REGION Network 34: CONVEYORS
   // FC71 = 0 IN + 0 OUT; FC72 = 0 IN + 1 OUT; FC73 = 0 IN + 2 OUT; FC74 = 0 IN + 3 OUT; FC75 = 0 IN + 4 OUT
   // FC76 = 1 IN + 0 OUT; FC77 = 1 IN + 1 OUT; FC78 = 1 IN + 2 OUT; FC79 = 1 IN + 3 OUT
   // FC80 = 2 IN + 0 OUT; FC81 = 2 IN + 1 OUT; FC82 = 2 IN + 2 OUT
   // FC83 = 3 IN + 0 OUT; FC84 = 3 IN + 1 OUT
   // FC85 = 4 IN + 0 OUT
   // FC86 = SPECIAL
   RUNG wire#powerrail
      Contact( "On" )
      wire#w1
      "FC31_ConveyorInverter"()
   END_RUNG
   RUNG wire#w1
      I_Contact( "On" )
      "FC32_ConveyorInverter_REV"()
   END_RUNG
   RUNG wire#w1
      { S7_Templates := "SrcType := Int" } EQ_Contact(in1 := "DB50_Config".Sel10_Conv, in2 := 16)
      "FC86_Conveyor_5_IN_3_OUT"()
   END_RUNG
   RUNG wire#w1
      { S7_Templates := "SrcType := Int" } EQ_Contact(in1 := "DB50_Config".Sel10_Conv, in2 := 1)
      "FC71_Conveyor_0_IN_0_OUT"()
   END_RUNG
   RUNG wire#w1
      { S7_Templates := "SrcType := Int" } EQ_Contact(in1 := "DB50_Config".Sel10_Conv, in2 := 2)
      "FC72_Conveyor_0_IN_1_OUT"()
   END_RUNG
   RUNG wire#w1
      { S7_Templates := "SrcType := Int" } EQ_Contact(in1 := "DB50_Config".Sel10_Conv, in2 := 7)
      wire#w2
      "FC77_Conveyor_1_IN_1_OUT"()
   END_RUNG
   RUNG wire#w2
      I_Contact( "On" )
      "FC78_Conveyor_1_IN_1_OUT_REVERSE"()
   END_RUNG
   RUNG wire#w1
      { S7_Templates := "SrcType := Int" } EQ_Contact(in1 := "DB50_Config".Sel10_Conv, in2 := 12)
      "FC82_Conveyor_2_IN_2_OUT"()
   END_RUNG
   // the same network as SCL:
   #_w1 := "On";
   IF #_w1 THEN "FC31_ConveyorInverter"(); END_IF;
   IF #_w1 AND NOT "On" THEN "FC32_ConveyorInverter_REV"(); END_IF;
   IF #_w1 AND ("DB50_Config".Sel10_Conv = 16) THEN "FC86_Conveyor_5_IN_3_OUT"(); END_IF;
   IF #_w1 AND ("DB50_Config".Sel10_Conv = 1) THEN "FC71_Conveyor_0_IN_0_OUT"(); END_IF;
   IF #_w1 AND ("DB50_Config".Sel10_Conv = 2) THEN "FC72_Conveyor_0_IN_1_OUT"(); END_IF;
   #_w2 := #_w1 AND ("DB50_Config".Sel10_Conv = 7);
   IF #_w2 THEN "FC77_Conveyor_1_IN_1_OUT"(); END_IF;
   IF #_w2 AND NOT "On" THEN "FC78_Conveyor_1_IN_1_OUT_REVERSE"(); END_IF;
   IF #_w1 AND ("DB50_Config".Sel10_Conv = 12) THEN "FC82_Conveyor_2_IN_2_OUT"(); END_IF;
END_REGION

REGION Network 35: BARRIERS
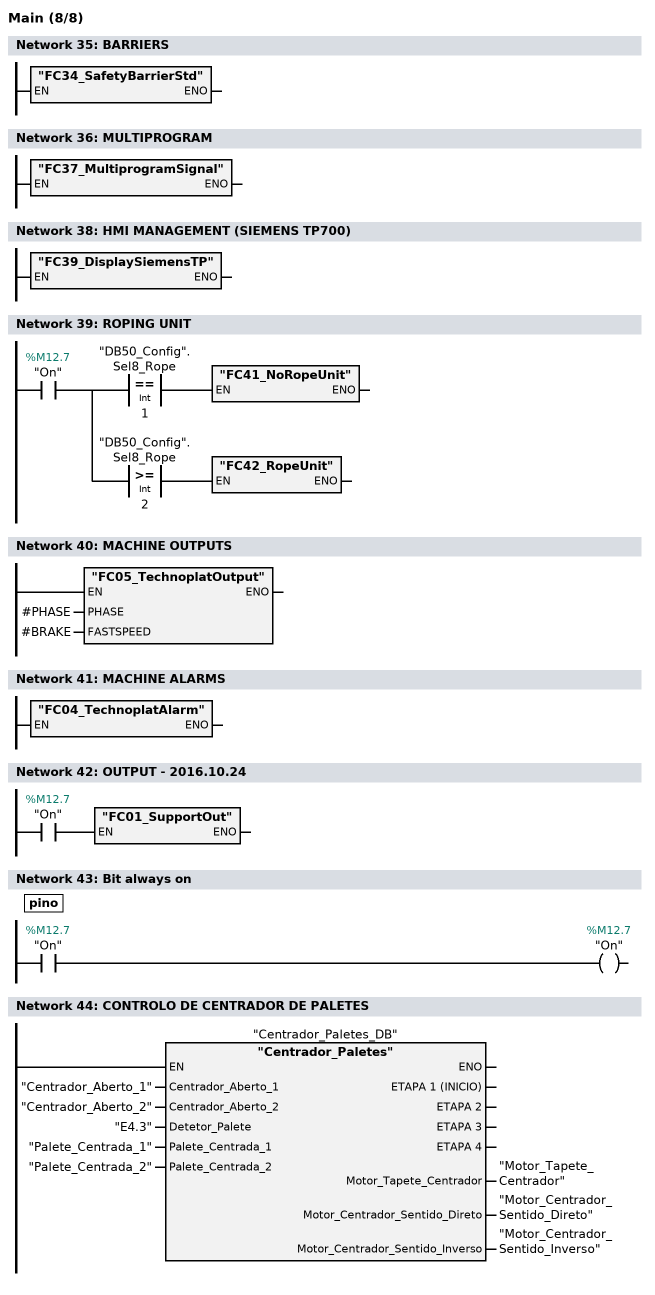
   RUNG wire#powerrail
      "FC34_SafetyBarrierStd"()
   END_RUNG
   // the same network as SCL:
   "FC34_SafetyBarrierStd"();
END_REGION

REGION Network 36: MULTIPROGRAM
   RUNG wire#powerrail
      "FC37_MultiprogramSignal"()
   END_RUNG
   // the same network as SCL:
   "FC37_MultiprogramSignal"();
END_REGION

REGION Network 37: Incomplete pallet
END_REGION

REGION Network 38: HMI MANAGEMENT (SIEMENS TP700)
   RUNG wire#powerrail
      "FC39_DisplaySiemensTP"()
   END_RUNG
   // the same network as SCL:
   "FC39_DisplaySiemensTP"();
END_REGION

REGION Network 39: ROPING UNIT
   RUNG wire#powerrail
      Contact( "On" )
      wire#w1
      { S7_Templates := "SrcType := Int" } EQ_Contact(in1 := "DB50_Config".Sel8_Rope, in2 := 1)
      "FC41_NoRopeUnit"()
   END_RUNG
   RUNG wire#w1
      { S7_Templates := "SrcType := Int" } GE_Contact(in1 := "DB50_Config".Sel8_Rope, in2 := 2)
      "FC42_RopeUnit"()
   END_RUNG
   // the same network as SCL:
   #_w1 := "On";
   IF "On" AND ("DB50_Config".Sel8_Rope = 1) THEN "FC41_NoRopeUnit"(); END_IF;
   IF #_w1 AND ("DB50_Config".Sel8_Rope >= 2) THEN "FC42_RopeUnit"(); END_IF;
END_REGION

REGION Network 40: MACHINE OUTPUTS
   RUNG wire#powerrail
      "FC05_TechnoplatOutput"(PHASE := #PHASE, FASTSPEED := #BRAKE)
   END_RUNG
   // the same network as SCL:
   "FC05_TechnoplatOutput"(PHASE := #PHASE, FASTSPEED := #BRAKE);
END_REGION

REGION Network 41: MACHINE ALARMS
   RUNG wire#powerrail
      "FC04_TechnoplatAlarm"()
   END_RUNG
   // the same network as SCL:
   "FC04_TechnoplatAlarm"();
END_REGION

REGION Network 42: OUTPUT - 2016.10.24
   RUNG wire#powerrail
      Contact( "On" )
      "FC01_SupportOut"()
   END_RUNG
   // the same network as SCL:
   IF "On" THEN "FC01_SupportOut"(); END_IF;
END_REGION

REGION Network 43: Bit always on
   Label( pino )
   RUNG wire#powerrail
      Contact( "On" )
      Coil( "On" )
   END_RUNG
   // the same network as SCL:
   pino:
   "On" := "On";
END_REGION

REGION Network 44: CONTROLO DE CENTRADOR DE PALETES
   RUNG wire#powerrail
      "Centrador_Paletes_DB"(Centrador_Aberto_1 := "Centrador_Aberto_1", Centrador_Aberto_2 := "Centrador_Aberto_2", Detetor_Palete := "E4.3", Palete_Centrada_1 := "Palete_Centrada_1", Palete_Centrada_2 := "Palete_Centrada_2", "ETAPA 1 (INICIO)" =>, "ETAPA 2" =>, "ETAPA 3" =>, "ETAPA 4" =>, Motor_Tapete_Centrador => "Motor_Tapete_Centrador", Motor_Centrador_Sentido_Direto => "Motor_Centrador_Sentido_Direto", Motor_Centrador_Sentido_Inverso => "Motor_Centrador_Sentido_Inverso")
   END_RUNG
   // the same network as SCL:
   "Centrador_Paletes_DB"(Centrador_Aberto_1 := "Centrador_Aberto_1",   // "Centrador_Paletes"
                          Centrador_Aberto_2 := "Centrador_Aberto_2",
                          Detetor_Palete := "E4.3",
                          Palete_Centrada_1 := "Palete_Centrada_1",
                          Palete_Centrada_2 := "Palete_Centrada_2",
                          Motor_Tapete_Centrador => "Motor_Tapete_Centrador",
                          Motor_Centrador_Sentido_Direto => "Motor_Centrador_Sentido_Direto",
                          Motor_Centrador_Sentido_Inverso => "Motor_Centrador_Sentido_Inverso");
END_REGION
END_ORGANIZATION_BLOCK

FUNCTION_BLOCK "Modbus"   // FB20, FBD
{ S7_Optimized_Access := 'FALSE' }
VERSION : 0.1
// stored: AutoNumber false, IsIECCheckEnabled false, SetENOAutomatically false, UDAEnableTagReadback false
   VAR_INPUT
      BAUDRATE : UDInt := 115200;
      HW_ID : PORT := 272;
      RESP_TO : UInt := 1000;
      CYCLIC_PROCESSING : Bool := true;
      MB_ADDR : UInt := 8;
      DATA_AD_R : UDInt := 40001;
      DATA_AD_W : UDInt := 40006;
      DATA_LEN_R : UInt := 5;
      DATA_LEN_W : UInt := 5;
      ReadOnly : Bool := 1;   // Read only (1)
   END_VAR
   VAR_OUTPUT
      ERROR : Bool;
      ERROR_INFO : Struct
         drive_number : USInt;
         "step" : USInt;
         STATUS : Word;
      END_STRUCT;
   END_VAR
   VAR_IN_OUT
      ReadDone_0 : Bool;   // Read done for prestretch board (1)
      DT_PTR_IN : Variant;
      DT_PTR_OUT : Variant;
   END_VAR
   VAR DB_SPECIFIC
      drive_index : USInt := 1;
      "step" : USInt := 0;
      REQ : Bool;
      extended_restart : Bool;
      start_internal : Bool;
   END_VAR
   VAR
      MB_COMM_LOAD_Instance { S7_SetPoint := 'True'} : MB_COMM_LOAD;
      MB_MASTER_Instance { S7_SetPoint := 'True'} : MB_MASTER;
   END_VAR
   VAR_TEMP
      _DONE : Bool;
      _ERROR : Bool;
      _STATUS : Word;
      _cyclic_processing : Bool;
   END_VAR
   VAR_TEMP   // added for the SCL form of the ladder/FBD networks
      _w1 : Bool;
      _w2 : Bool;
      _w3 : Bool;
   END_VAR
BEGIN

REGION Network 1: First cycle
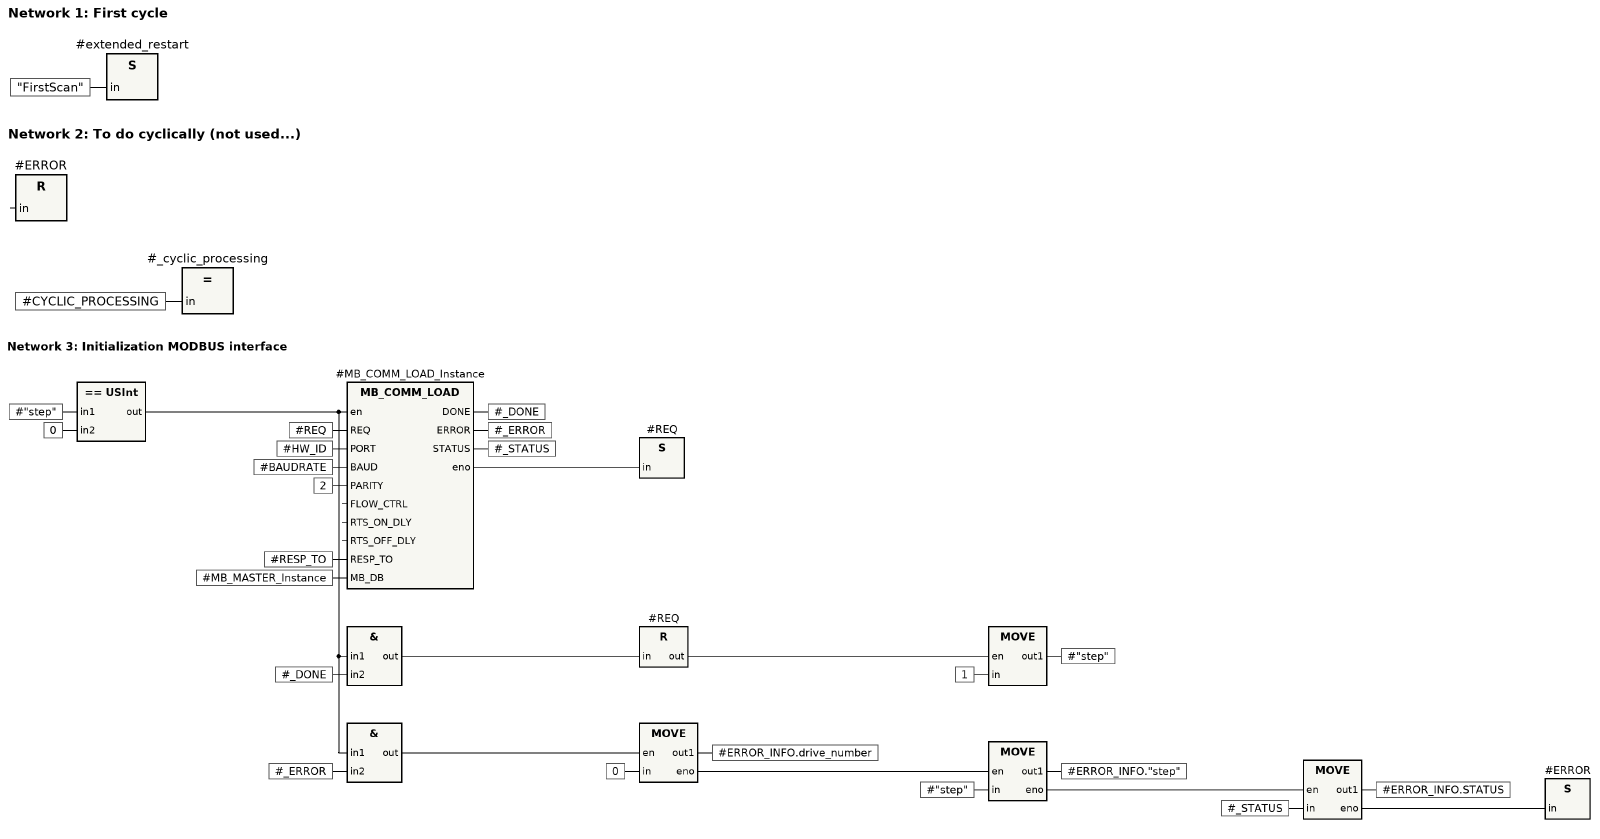
   IF "FirstScan" THEN #extended_restart := TRUE; END_IF;
END_REGION

REGION Network 2: To do cyclically (not used...)
   #ERROR := FALSE;
   #_cyclic_processing := #CYCLIC_PROCESSING;
END_REGION

REGION Network 3: Initialization MODBUS interface
   // ENO of a box is taken as its EN; it also drops when the box reports an error
   #_w1 := #"step" = 0;
   #MB_COMM_LOAD_Instance(EN := #_w1,   // MB_COMM_LOAD
                          REQ := #REQ,
                          PORT := #HW_ID,
                          BAUD := #BAUDRATE,
                          PARITY := 2,
                          RESP_TO := #RESP_TO,
                          MB_DB := #MB_MASTER_Instance,
                          DONE => #_DONE,
                          ERROR => #_ERROR,
                          STATUS => #_STATUS,
                          ENO => #_w2);
   IF #_w2 THEN #REQ := TRUE; END_IF;
   IF #_w1 AND #_DONE THEN
       #REQ := FALSE;
       #"step" := 1;
   END_IF;
   IF #_w1 AND #_ERROR THEN
       #ERROR_INFO.drive_number := 0;
       #ERROR_INFO."step" := #"step";
       #ERROR_INFO.STATUS := #_STATUS;
       #ERROR := TRUE;
   END_IF;
END_REGION

REGION Network 4: READ
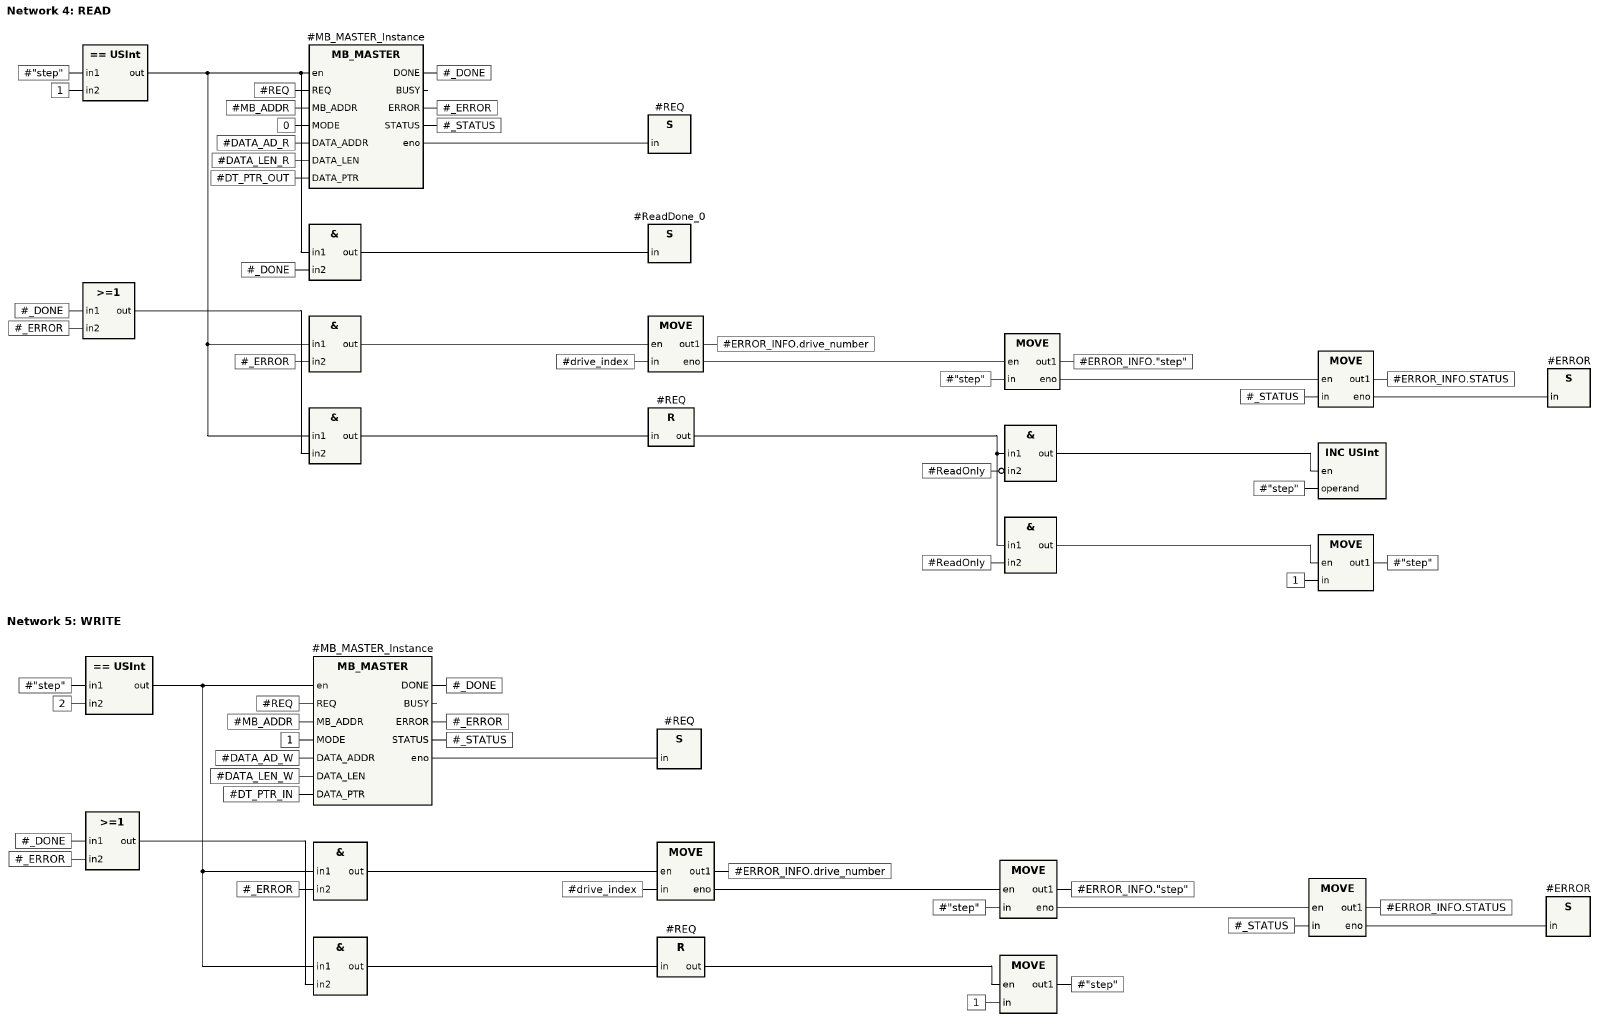
   // ENO of a box is taken as its EN; it also drops when the box reports an error
   #_w1 := #"step" = 1;
   #MB_MASTER_Instance(EN := #_w1,   // MB_MASTER
                       REQ := #REQ,
                       MB_ADDR := #MB_ADDR,
                       MODE := 0,
                       DATA_ADDR := #DATA_AD_R,
                       DATA_LEN := #DATA_LEN_R,
                       DATA_PTR := #DT_PTR_OUT,
                       DONE => #_DONE,
                       ERROR => #_ERROR,
                       STATUS => #_STATUS,
                       ENO => #_w2);
   IF #_w2 THEN #REQ := TRUE; END_IF;
   IF #_w1 AND #_DONE THEN #ReadDone_0 := TRUE; END_IF;
   IF #_w1 AND #_ERROR THEN
       #ERROR_INFO.drive_number := #drive_index;
       #ERROR_INFO."step" := #"step";
       #ERROR_INFO.STATUS := #_STATUS;
       #ERROR := TRUE;
   END_IF;
   #_w3 := #_w1 AND (#_DONE OR #_ERROR);
   IF #_w3 THEN #REQ := FALSE; END_IF;
   IF #_w3 AND NOT #ReadOnly THEN #"step" := #"step" + 1; END_IF;
   IF #_w3 AND #ReadOnly THEN #"step" := 1; END_IF;
END_REGION

REGION Network 5: WRITE
   // ENO of a box is taken as its EN; it also drops when the box reports an error
   #_w1 := #"step" = 2;
   #MB_MASTER_Instance(EN := #_w1,   // MB_MASTER
                       REQ := #REQ,
                       MB_ADDR := #MB_ADDR,
                       MODE := 1,
                       DATA_ADDR := #DATA_AD_W,
                       DATA_LEN := #DATA_LEN_W,
                       DATA_PTR := #DT_PTR_IN,
                       DONE => #_DONE,
                       ERROR => #_ERROR,
                       STATUS => #_STATUS,
                       ENO => #_w2);
   IF #_w2 THEN #REQ := TRUE; END_IF;
   IF #_w1 AND #_ERROR THEN
       #ERROR_INFO.drive_number := #drive_index;
       #ERROR_INFO."step" := #"step";
       #ERROR_INFO.STATUS := #_STATUS;
       #ERROR := TRUE;
   END_IF;
   IF #_w1 AND (#_DONE OR #_ERROR) THEN
       #REQ := FALSE;
       #"step" := 1;
   END_IF;
END_REGION
END_FUNCTION_BLOCK

FUNCTION "FC81_Optional" : Void   // FC81, LAD
TITLE = Optional
{ S7_Optimized_Access := 'TRUE' }
VERSION : 0.1
// stored: AutoNumber false, IsIECCheckEnabled false, SetENOAutomatically false, UDAEnableTagReadback false
BEGIN

REGION Network 1: Signal Automatic
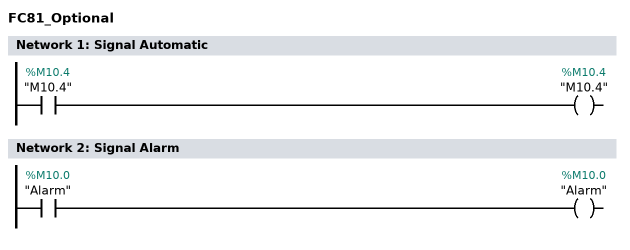
   RUNG wire#powerrail
      Contact( "M10.4" )
      Coil( "M10.4" )
   END_RUNG
   // the same network as SCL:
   "M10.4" := "M10.4";
END_REGION

REGION Network 2: Signal Alarm
   RUNG wire#powerrail
      Contact( "Alarm" )
      Coil( "Alarm" )
   END_RUNG
   // the same network as SCL:
   "Alarm" := "Alarm";
END_REGION
END_FUNCTION

FUNCTION "FC90_PageManagement" : Void   // FC90, LAD
{ S7_Optimized_Access := 'FALSE' }
VERSION : 0.1
// stored: AutoNumber false, IsIECCheckEnabled false, SetENOAutomatically false, UDAEnableTagReadback false
   VAR_TEMP
      CurrentPage : Int;
      PageBkwRequest : Int;
      PageFwRequest : Int;
   END_VAR
   VAR_TEMP   // added for the SCL form of the ladder/FBD networks
      _w1 : Bool;
   END_VAR
BEGIN

REGION Network 1
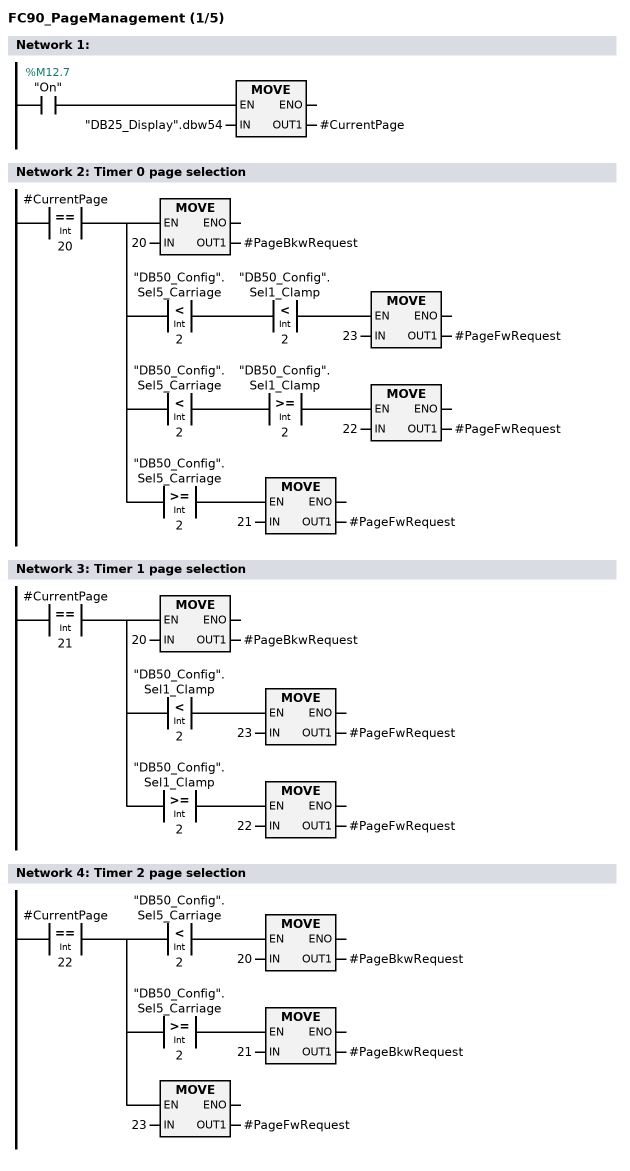
   RUNG wire#powerrail
      Contact( "On" )
      { S7_GenerateENO := "TRUE" } Move(in := "DB25_Display".dbw54, out1 => #CurrentPage)
   END_RUNG
   // the same network as SCL:
   IF "On" THEN #CurrentPage := "DB25_Display".dbw54; END_IF;
END_REGION

REGION Network 2: Timer 0 page selection
   RUNG wire#powerrail
      { S7_Templates := "SrcType := Int" } EQ_Contact(in1 := #CurrentPage, in2 := 20)
      wire#w1
      { S7_GenerateENO := "TRUE" } Move(in := 20, out1 => #PageBkwRequest)
   END_RUNG
   RUNG wire#w1
      { S7_Templates := "SrcType := Int" } LT_Contact(in1 := "DB50_Config".Sel5_Carriage, in2 := 2)
      { S7_Templates := "SrcType := Int" } LT_Contact(in1 := "DB50_Config".Sel1_Clamp, in2 := 2)
      { S7_GenerateENO := "TRUE" } Move(in := 23, out1 => #PageFwRequest)
   END_RUNG
   RUNG wire#w1
      { S7_Templates := "SrcType := Int" } LT_Contact(in1 := "DB50_Config".Sel5_Carriage, in2 := 2)
      { S7_Templates := "SrcType := Int" } GE_Contact(in1 := "DB50_Config".Sel1_Clamp, in2 := 2)
      { S7_GenerateENO := "TRUE" } Move(in := 22, out1 => #PageFwRequest)
   END_RUNG
   RUNG wire#w1
      { S7_Templates := "SrcType := Int" } GE_Contact(in1 := "DB50_Config".Sel5_Carriage, in2 := 2)
      { S7_GenerateENO := "TRUE" } Move(in := 21, out1 => #PageFwRequest)
   END_RUNG
   // the same network as SCL:
   #_w1 := #CurrentPage = 20;
   IF #_w1 THEN #PageBkwRequest := 20; END_IF;
   IF #_w1 AND ("DB50_Config".Sel5_Carriage < 2) AND ("DB50_Config".Sel1_Clamp < 2) THEN
       #PageFwRequest := 23;
   END_IF;
   IF #_w1 AND ("DB50_Config".Sel5_Carriage < 2) AND ("DB50_Config".Sel1_Clamp >= 2) THEN
       #PageFwRequest := 22;
   END_IF;
   IF #_w1 AND ("DB50_Config".Sel5_Carriage >= 2) THEN #PageFwRequest := 21; END_IF;
END_REGION

REGION Network 3: Timer 1 page selection
   RUNG wire#powerrail
      { S7_Templates := "SrcType := Int" } EQ_Contact(in1 := #CurrentPage, in2 := 21)
      wire#w1
      { S7_GenerateENO := "TRUE" } Move(in := 20, out1 => #PageBkwRequest)
   END_RUNG
   RUNG wire#w1
      { S7_Templates := "SrcType := Int" } LT_Contact(in1 := "DB50_Config".Sel1_Clamp, in2 := 2)
      { S7_GenerateENO := "TRUE" } Move(in := 23, out1 => #PageFwRequest)
   END_RUNG
   RUNG wire#w1
      { S7_Templates := "SrcType := Int" } GE_Contact(in1 := "DB50_Config".Sel1_Clamp, in2 := 2)
      { S7_GenerateENO := "TRUE" } Move(in := 22, out1 => #PageFwRequest)
   END_RUNG
   // the same network as SCL:
   #_w1 := #CurrentPage = 21;
   IF #_w1 THEN #PageBkwRequest := 20; END_IF;
   IF #_w1 AND ("DB50_Config".Sel1_Clamp < 2) THEN #PageFwRequest := 23; END_IF;
   IF #_w1 AND ("DB50_Config".Sel1_Clamp >= 2) THEN #PageFwRequest := 22; END_IF;
END_REGION

REGION Network 4: Timer 2 page selection
   RUNG wire#powerrail
      { S7_Templates := "SrcType := Int" } EQ_Contact(in1 := #CurrentPage, in2 := 22)
      wire#w1
      { S7_Templates := "SrcType := Int" } LT_Contact(in1 := "DB50_Config".Sel5_Carriage, in2 := 2)
      { S7_GenerateENO := "TRUE" } Move(in := 20, out1 => #PageBkwRequest)
   END_RUNG
   RUNG wire#w1
      { S7_Templates := "SrcType := Int" } GE_Contact(in1 := "DB50_Config".Sel5_Carriage, in2 := 2)
      { S7_GenerateENO := "TRUE" } Move(in := 21, out1 => #PageBkwRequest)
   END_RUNG
   RUNG wire#w1
      { S7_GenerateENO := "TRUE" } Move(in := 23, out1 => #PageFwRequest)
   END_RUNG
   // the same network as SCL:
   #_w1 := #CurrentPage = 22;
   IF #_w1 AND ("DB50_Config".Sel5_Carriage < 2) THEN #PageBkwRequest := 20; END_IF;
   IF #_w1 AND ("DB50_Config".Sel5_Carriage >= 2) THEN #PageBkwRequest := 21; END_IF;
   IF #_w1 THEN #PageFwRequest := 23; END_IF;
END_REGION

REGION Network 5: Timer 3 page selection
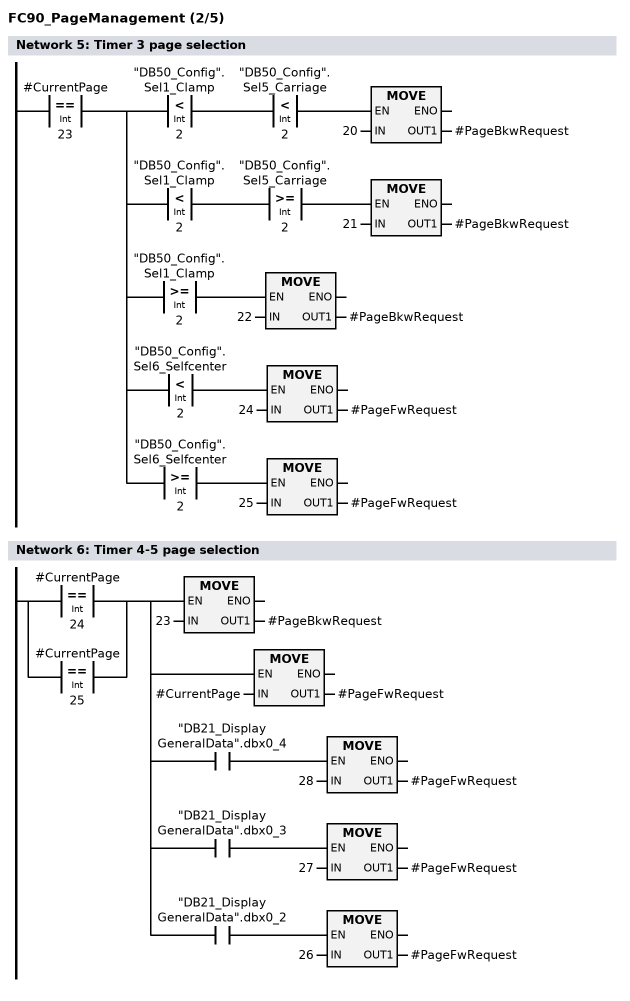
   RUNG wire#powerrail
      { S7_Templates := "SrcType := Int" } EQ_Contact(in1 := #CurrentPage, in2 := 23)
      wire#w1
      { S7_Templates := "SrcType := Int" } LT_Contact(in1 := "DB50_Config".Sel1_Clamp, in2 := 2)
      { S7_Templates := "SrcType := Int" } LT_Contact(in1 := "DB50_Config".Sel5_Carriage, in2 := 2)
      { S7_GenerateENO := "TRUE" } Move(in := 20, out1 => #PageBkwRequest)
   END_RUNG
   RUNG wire#w1
      { S7_Templates := "SrcType := Int" } LT_Contact(in1 := "DB50_Config".Sel1_Clamp, in2 := 2)
      { S7_Templates := "SrcType := Int" } GE_Contact(in1 := "DB50_Config".Sel5_Carriage, in2 := 2)
      { S7_GenerateENO := "TRUE" } Move(in := 21, out1 => #PageBkwRequest)
   END_RUNG
   RUNG wire#w1
      { S7_Templates := "SrcType := Int" } GE_Contact(in1 := "DB50_Config".Sel1_Clamp, in2 := 2)
      { S7_GenerateENO := "TRUE" } Move(in := 22, out1 => #PageBkwRequest)
   END_RUNG
   RUNG wire#w1
      { S7_Templates := "SrcType := Int" } LT_Contact(in1 := "DB50_Config".Sel6_Selfcenter, in2 := 2)
      { S7_GenerateENO := "TRUE" } Move(in := 24, out1 => #PageFwRequest)
   END_RUNG
   RUNG wire#w1
      { S7_Templates := "SrcType := Int" } GE_Contact(in1 := "DB50_Config".Sel6_Selfcenter, in2 := 2)
      { S7_GenerateENO := "TRUE" } Move(in := 25, out1 => #PageFwRequest)
   END_RUNG
   // the same network as SCL:
   #_w1 := #CurrentPage = 23;
   IF #_w1 AND ("DB50_Config".Sel1_Clamp < 2) AND ("DB50_Config".Sel5_Carriage < 2) THEN
       #PageBkwRequest := 20;
   END_IF;
   IF #_w1 AND ("DB50_Config".Sel1_Clamp < 2) AND ("DB50_Config".Sel5_Carriage >= 2) THEN
       #PageBkwRequest := 21;
   END_IF;
   IF #_w1 AND ("DB50_Config".Sel1_Clamp >= 2) THEN #PageBkwRequest := 22; END_IF;
   IF #_w1 AND ("DB50_Config".Sel6_Selfcenter < 2) THEN #PageFwRequest := 24; END_IF;
   IF #_w1 AND ("DB50_Config".Sel6_Selfcenter >= 2) THEN #PageFwRequest := 25; END_IF;
END_REGION

REGION Network 6: Timer 4-5 page selection
   RUNG wire#powerrail
      { S7_Templates := "SrcType := Int" } EQ_Contact(in1 := #CurrentPage, in2 := 24)
      wire#w1
      { S7_GenerateENO := "TRUE" } Move(in := 23, out1 => #PageBkwRequest)
   END_RUNG
   RUNG wire#powerrail
      { S7_Templates := "SrcType := Int" } EQ_Contact(in1 := #CurrentPage, in2 := 25)
   END_RUNG wire#w1
   RUNG wire#w1
      { S7_GenerateENO := "TRUE" } Move(in := #CurrentPage, out1 => #PageFwRequest)
   END_RUNG
   RUNG wire#w1
      Contact( "DB21_DisplayGeneralData".dbx0_4 )
      { S7_GenerateENO := "TRUE" } Move(in := 28, out1 => #PageFwRequest)
   END_RUNG
   RUNG wire#w1
      Contact( "DB21_DisplayGeneralData".dbx0_3 )
      { S7_GenerateENO := "TRUE" } Move(in := 27, out1 => #PageFwRequest)
   END_RUNG
   RUNG wire#w1
      Contact( "DB21_DisplayGeneralData".dbx0_2 )
      { S7_GenerateENO := "TRUE" } Move(in := 26, out1 => #PageFwRequest)
   END_RUNG
   // the same network as SCL:
   #_w1 := (#CurrentPage = 24) OR (#CurrentPage = 25);
   IF #_w1 THEN
       #PageBkwRequest := 23;
       #PageFwRequest := #CurrentPage;
   END_IF;
   IF #_w1 AND "DB21_DisplayGeneralData".dbx0_4 THEN #PageFwRequest := 28; END_IF;
   IF #_w1 AND "DB21_DisplayGeneralData".dbx0_3 THEN #PageFwRequest := 27; END_IF;
   IF #_w1 AND "DB21_DisplayGeneralData".dbx0_2 THEN #PageFwRequest := 26; END_IF;
END_REGION

REGION Network 7: Timer 6 page selection
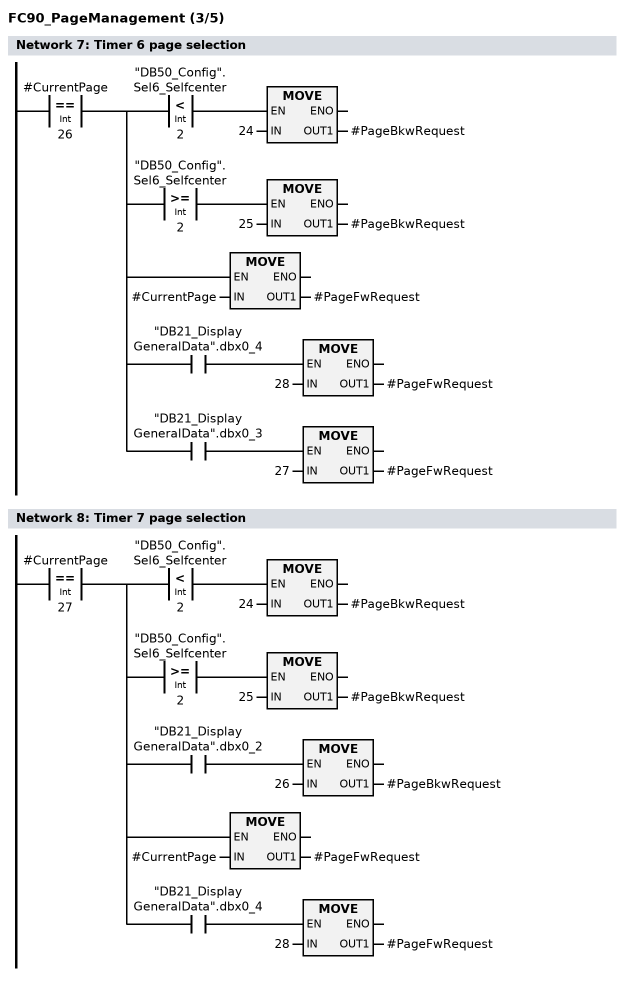
   RUNG wire#powerrail
      { S7_Templates := "SrcType := Int" } EQ_Contact(in1 := #CurrentPage, in2 := 26)
      wire#w1
      { S7_Templates := "SrcType := Int" } LT_Contact(in1 := "DB50_Config".Sel6_Selfcenter, in2 := 2)
      { S7_GenerateENO := "TRUE" } Move(in := 24, out1 => #PageBkwRequest)
   END_RUNG
   RUNG wire#w1
      { S7_Templates := "SrcType := Int" } GE_Contact(in1 := "DB50_Config".Sel6_Selfcenter, in2 := 2)
      { S7_GenerateENO := "TRUE" } Move(in := 25, out1 => #PageBkwRequest)
   END_RUNG
   RUNG wire#w1
      { S7_GenerateENO := "TRUE" } Move(in := #CurrentPage, out1 => #PageFwRequest)
   END_RUNG
   RUNG wire#w1
      Contact( "DB21_DisplayGeneralData".dbx0_4 )
      { S7_GenerateENO := "TRUE" } Move(in := 28, out1 => #PageFwRequest)
   END_RUNG
   RUNG wire#w1
      Contact( "DB21_DisplayGeneralData".dbx0_3 )
      { S7_GenerateENO := "TRUE" } Move(in := 27, out1 => #PageFwRequest)
   END_RUNG
   // the same network as SCL:
   #_w1 := #CurrentPage = 26;
   IF #_w1 AND ("DB50_Config".Sel6_Selfcenter < 2) THEN #PageBkwRequest := 24; END_IF;
   IF #_w1 AND ("DB50_Config".Sel6_Selfcenter >= 2) THEN #PageBkwRequest := 25; END_IF;
   IF #_w1 THEN #PageFwRequest := #CurrentPage; END_IF;
   IF #_w1 AND "DB21_DisplayGeneralData".dbx0_4 THEN #PageFwRequest := 28; END_IF;
   IF #_w1 AND "DB21_DisplayGeneralData".dbx0_3 THEN #PageFwRequest := 27; END_IF;
END_REGION

REGION Network 8: Timer 7 page selection
   RUNG wire#powerrail
      { S7_Templates := "SrcType := Int" } EQ_Contact(in1 := #CurrentPage, in2 := 27)
      wire#w1
      { S7_Templates := "SrcType := Int" } LT_Contact(in1 := "DB50_Config".Sel6_Selfcenter, in2 := 2)
      { S7_GenerateENO := "TRUE" } Move(in := 24, out1 => #PageBkwRequest)
   END_RUNG
   RUNG wire#w1
      { S7_Templates := "SrcType := Int" } GE_Contact(in1 := "DB50_Config".Sel6_Selfcenter, in2 := 2)
      { S7_GenerateENO := "TRUE" } Move(in := 25, out1 => #PageBkwRequest)
   END_RUNG
   RUNG wire#w1
      Contact( "DB21_DisplayGeneralData".dbx0_2 )
      { S7_GenerateENO := "TRUE" } Move(in := 26, out1 => #PageBkwRequest)
   END_RUNG
   RUNG wire#w1
      { S7_GenerateENO := "TRUE" } Move(in := #CurrentPage, out1 => #PageFwRequest)
   END_RUNG
   RUNG wire#w1
      Contact( "DB21_DisplayGeneralData".dbx0_4 )
      { S7_GenerateENO := "TRUE" } Move(in := 28, out1 => #PageFwRequest)
   END_RUNG
   // the same network as SCL:
   #_w1 := #CurrentPage = 27;
   IF #_w1 AND ("DB50_Config".Sel6_Selfcenter < 2) THEN #PageBkwRequest := 24; END_IF;
   IF #_w1 AND ("DB50_Config".Sel6_Selfcenter >= 2) THEN #PageBkwRequest := 25; END_IF;
   IF #_w1 AND "DB21_DisplayGeneralData".dbx0_2 THEN #PageBkwRequest := 26; END_IF;
   IF #_w1 THEN #PageFwRequest := #CurrentPage; END_IF;
   IF #_w1 AND "DB21_DisplayGeneralData".dbx0_4 THEN #PageFwRequest := 28; END_IF;
END_REGION

REGION Network 9: Timer 8 page selection
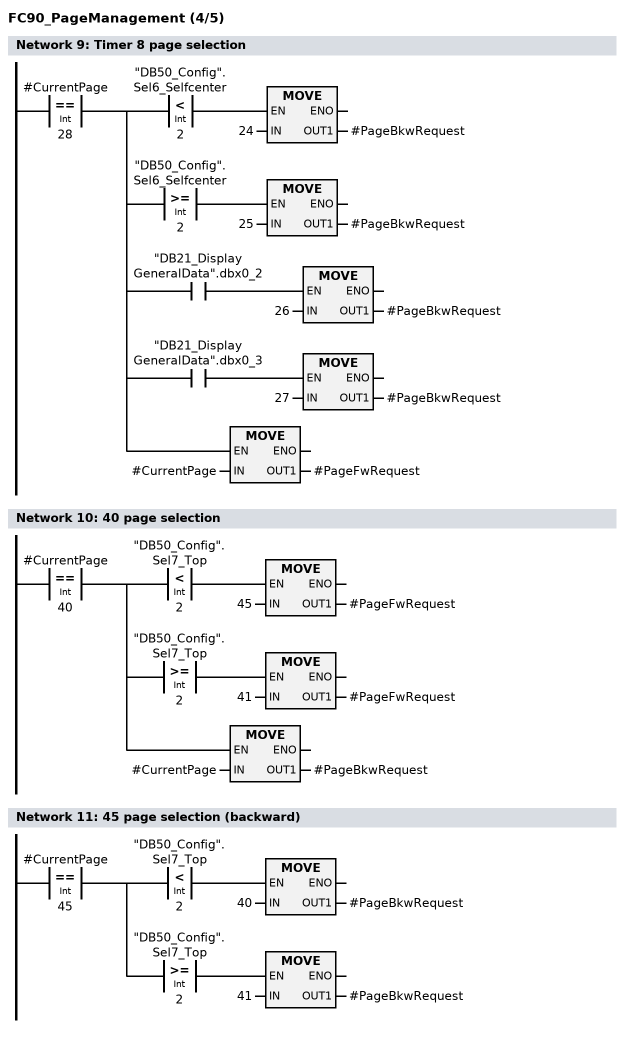
   RUNG wire#powerrail
      { S7_Templates := "SrcType := Int" } EQ_Contact(in1 := #CurrentPage, in2 := 28)
      wire#w1
      { S7_Templates := "SrcType := Int" } LT_Contact(in1 := "DB50_Config".Sel6_Selfcenter, in2 := 2)
      { S7_GenerateENO := "TRUE" } Move(in := 24, out1 => #PageBkwRequest)
   END_RUNG
   RUNG wire#w1
      { S7_Templates := "SrcType := Int" } GE_Contact(in1 := "DB50_Config".Sel6_Selfcenter, in2 := 2)
      { S7_GenerateENO := "TRUE" } Move(in := 25, out1 => #PageBkwRequest)
   END_RUNG
   RUNG wire#w1
      Contact( "DB21_DisplayGeneralData".dbx0_2 )
      { S7_GenerateENO := "TRUE" } Move(in := 26, out1 => #PageBkwRequest)
   END_RUNG
   RUNG wire#w1
      Contact( "DB21_DisplayGeneralData".dbx0_3 )
      { S7_GenerateENO := "TRUE" } Move(in := 27, out1 => #PageBkwRequest)
   END_RUNG
   RUNG wire#w1
      { S7_GenerateENO := "TRUE" } Move(in := #CurrentPage, out1 => #PageFwRequest)
   END_RUNG
   // the same network as SCL:
   #_w1 := #CurrentPage = 28;
   IF #_w1 AND ("DB50_Config".Sel6_Selfcenter < 2) THEN #PageBkwRequest := 24; END_IF;
   IF #_w1 AND ("DB50_Config".Sel6_Selfcenter >= 2) THEN #PageBkwRequest := 25; END_IF;
   IF #_w1 AND "DB21_DisplayGeneralData".dbx0_2 THEN #PageBkwRequest := 26; END_IF;
   IF #_w1 AND "DB21_DisplayGeneralData".dbx0_3 THEN #PageBkwRequest := 27; END_IF;
   IF #_w1 THEN #PageFwRequest := #CurrentPage; END_IF;
END_REGION

REGION Network 10: 40 page selection
   RUNG wire#powerrail
      { S7_Templates := "SrcType := Int" } EQ_Contact(in1 := #CurrentPage, in2 := 40)
      wire#w1
      { S7_Templates := "SrcType := Int" } LT_Contact(in1 := "DB50_Config".Sel7_Top, in2 := 2)
      { S7_GenerateENO := "TRUE" } Move(in := 45, out1 => #PageFwRequest)
   END_RUNG
   RUNG wire#w1
      { S7_Templates := "SrcType := Int" } GE_Contact(in1 := "DB50_Config".Sel7_Top, in2 := 2)
      { S7_GenerateENO := "TRUE" } Move(in := 41, out1 => #PageFwRequest)
   END_RUNG
   RUNG wire#w1
      { S7_GenerateENO := "TRUE" } Move(in := #CurrentPage, out1 => #PageBkwRequest)
   END_RUNG
   // the same network as SCL:
   #_w1 := #CurrentPage = 40;
   IF #_w1 AND ("DB50_Config".Sel7_Top < 2) THEN #PageFwRequest := 45; END_IF;
   IF #_w1 AND ("DB50_Config".Sel7_Top >= 2) THEN #PageFwRequest := 41; END_IF;
   IF #_w1 THEN #PageBkwRequest := #CurrentPage; END_IF;
END_REGION

REGION Network 11: 45 page selection (backward)
   RUNG wire#powerrail
      { S7_Templates := "SrcType := Int" } EQ_Contact(in1 := #CurrentPage, in2 := 45)
      wire#w1
      { S7_Templates := "SrcType := Int" } LT_Contact(in1 := "DB50_Config".Sel7_Top, in2 := 2)
      { S7_GenerateENO := "TRUE" } Move(in := 40, out1 => #PageBkwRequest)
   END_RUNG
   RUNG wire#w1
      { S7_Templates := "SrcType := Int" } GE_Contact(in1 := "DB50_Config".Sel7_Top, in2 := 2)
      { S7_GenerateENO := "TRUE" } Move(in := 41, out1 => #PageBkwRequest)
   END_RUNG
   // the same network as SCL:
   #_w1 := #CurrentPage = 45;
   IF #_w1 AND ("DB50_Config".Sel7_Top < 2) THEN #PageBkwRequest := 40; END_IF;
   IF #_w1 AND ("DB50_Config".Sel7_Top >= 2) THEN #PageBkwRequest := 41; END_IF;
END_REGION

REGION Network 12
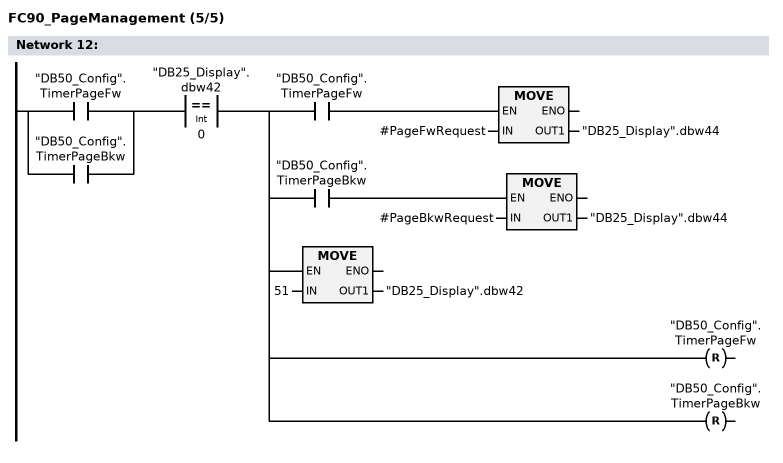
   RUNG wire#powerrail
      Contact( "DB50_Config".TimerPageFw )
      wire#w1
      { S7_Templates := "SrcType := Int" } EQ_Contact(in1 := "DB25_Display".dbw42, in2 := 0)
      wire#w2
      Contact( "DB50_Config".TimerPageFw )
      { S7_GenerateENO := "TRUE" } Move(in := #PageFwRequest, out1 => "DB25_Display".dbw44)
   END_RUNG
   RUNG wire#powerrail
      Contact( "DB50_Config".TimerPageBkw )
   END_RUNG wire#w1
   RUNG wire#w2
      Contact( "DB50_Config".TimerPageBkw )
      { S7_GenerateENO := "TRUE" } Move(in := #PageBkwRequest, out1 => "DB25_Display".dbw44)
   END_RUNG
   RUNG wire#w2
      { S7_GenerateENO := "TRUE" } Move(in := 51, out1 => "DB25_Display".dbw42)
   END_RUNG
   RUNG wire#w2
      R_Coil( "DB50_Config".TimerPageFw )
   END_RUNG
   RUNG wire#w2
      R_Coil( "DB50_Config".TimerPageBkw )
   END_RUNG
   // the same network as SCL:
   #_w1 := ("DB50_Config".TimerPageFw OR "DB50_Config".TimerPageBkw) AND ("DB25_Display".dbw42 = 0);
   IF #_w1 AND "DB50_Config".TimerPageFw THEN "DB25_Display".dbw44 := #PageFwRequest; END_IF;
   IF #_w1 AND "DB50_Config".TimerPageBkw THEN "DB25_Display".dbw44 := #PageBkwRequest; END_IF;
   IF #_w1 THEN
       "DB25_Display".dbw42 := 51;
       "DB50_Config".TimerPageFw := FALSE;
       "DB50_Config".TimerPageBkw := FALSE;
   END_IF;
END_REGION
END_FUNCTION

FUNCTION "FC00_SupportIn" : Void   // FC0, LAD
TITLE = Input support memory
{ S7_Optimized_Access := 'FALSE' }
AUTHOR : Robopac
VERSION : 0.0
// stored: AutoNumber false, IsIECCheckEnabled false, SetENOAutomatically false, UDAEnableTagReadback false
   VAR_TEMP
      AC1 : Int;
      AC2 : Int;
   END_VAR
BEGIN

REGION Network 1: STANDARD
END_REGION

REGION Network 2: Pressure switch (Technoplat)
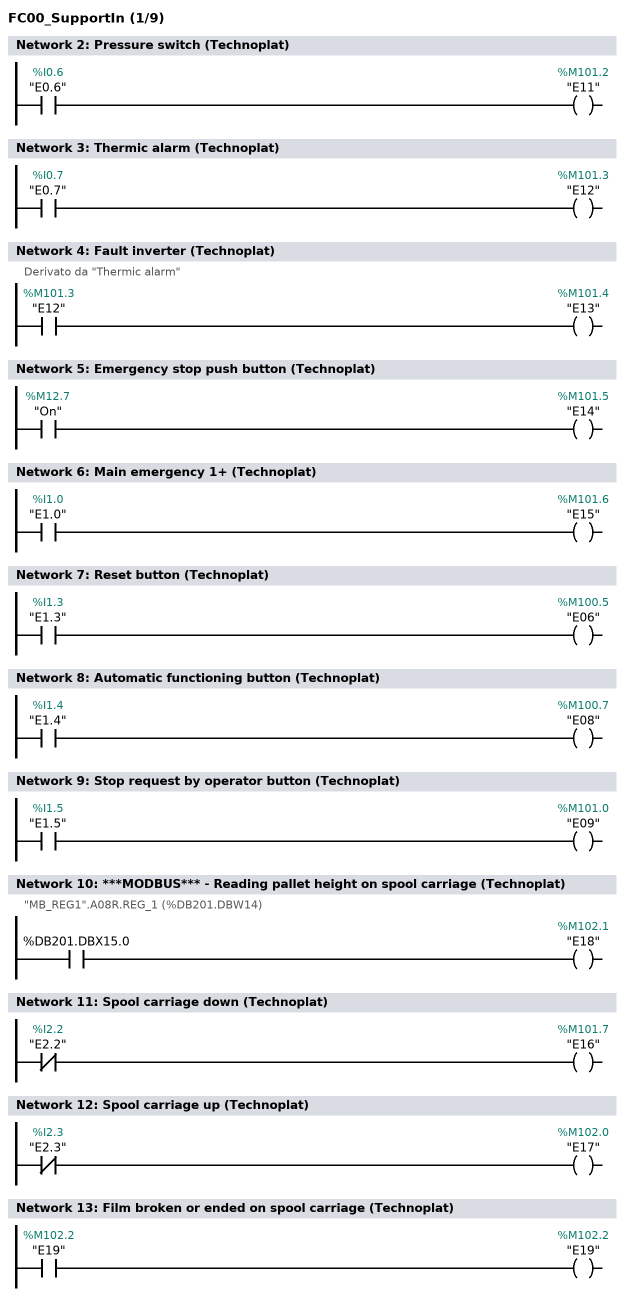
   RUNG wire#powerrail
      Contact( "E0.6" )
      Coil( "E11" )
   END_RUNG
   // the same network as SCL:
   "E11" := "E0.6";
END_REGION

REGION Network 3: Thermic alarm (Technoplat)
   RUNG wire#powerrail
      Contact( "E0.7" )
      Coil( "E12" )
   END_RUNG
   // the same network as SCL:
   "E12" := "E0.7";
END_REGION

REGION Network 4: Fault inverter (Technoplat)
   // Derivato da "Thermic alarm"
   RUNG wire#powerrail
      Contact( "E12" )
      Coil( "E13" )
   END_RUNG
   // the same network as SCL:
   "E13" := "E12";
END_REGION

REGION Network 5: Emergency stop push button (Technoplat)
   RUNG wire#powerrail
      Contact( "On" )
      Coil( "E14" )
   END_RUNG
   // the same network as SCL:
   "E14" := "On";
END_REGION

REGION Network 6: Main emergency 1+ (Technoplat)
   RUNG wire#powerrail
      Contact( "E1.0" )
      Coil( "E15" )
   END_RUNG
   // the same network as SCL:
   "E15" := "E1.0";
END_REGION

REGION Network 7: Reset button (Technoplat)
   RUNG wire#powerrail
      Contact( "E1.3" )
      Coil( "E06" )
   END_RUNG
   // the same network as SCL:
   "E06" := "E1.3";
END_REGION

REGION Network 8: Automatic functioning button (Technoplat)
   RUNG wire#powerrail
      Contact( "E1.4" )
      Coil( "E08" )
   END_RUNG
   // the same network as SCL:
   "E08" := "E1.4";
END_REGION

REGION Network 9: Stop request by operator button (Technoplat)
   RUNG wire#powerrail
      Contact( "E1.5" )
      Coil( "E09" )
   END_RUNG
   // the same network as SCL:
   "E09" := "E1.5";
END_REGION

REGION Network 10: ***MODBUS*** - Reading pallet height on spool carriage (Technoplat)
   // "MB_REG1".A08R.REG_1 (%DB201.DBW14)
   RUNG wire#powerrail
      Contact( %DB201.DBX15.0 )
      Coil( "E18" )
   END_RUNG
   // the same network as SCL:
   "E18" := %DB201.DBX15.0;
END_REGION

REGION Network 11: Spool carriage down (Technoplat)
   RUNG wire#powerrail
      I_Contact( "E2.2" )
      Coil( "E16" )
   END_RUNG
   // the same network as SCL:
   "E16" := NOT "E2.2";
END_REGION

REGION Network 12: Spool carriage up (Technoplat)
   RUNG wire#powerrail
      I_Contact( "E2.3" )
      Coil( "E17" )
   END_RUNG
   // the same network as SCL:
   "E17" := NOT "E2.3";
END_REGION

REGION Network 13: Film broken or ended on spool carriage (Technoplat)
   RUNG wire#powerrail
      Contact( "E19" )
      Coil( "E19" )
   END_RUNG
   // the same network as SCL:
   "E19" := "E19";
END_REGION

REGION Network 14: Cutting and welding unit backward (Claw clamp)
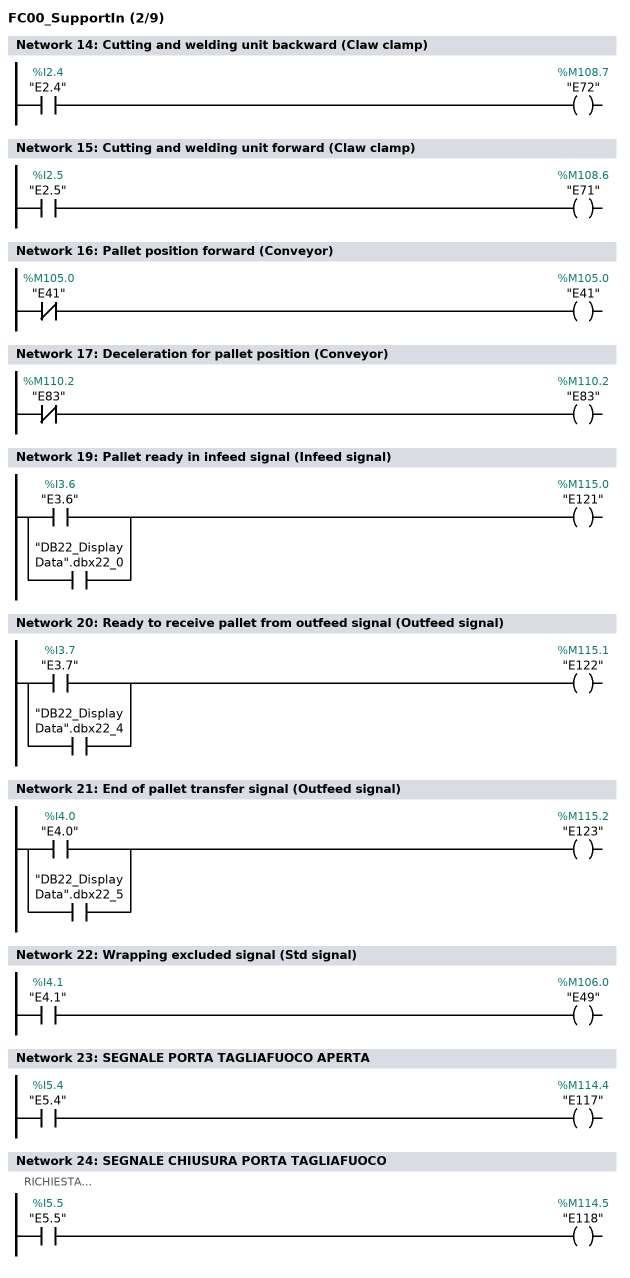
   RUNG wire#powerrail
      Contact( "E2.4" )
      Coil( "E72" )
   END_RUNG
   // the same network as SCL:
   "E72" := "E2.4";
END_REGION

REGION Network 15: Cutting and welding unit forward (Claw clamp)
   RUNG wire#powerrail
      Contact( "E2.5" )
      Coil( "E71" )
   END_RUNG
   // the same network as SCL:
   "E71" := "E2.5";
END_REGION

REGION Network 16: Pallet position forward (Conveyor)
   RUNG wire#powerrail
      I_Contact( "E41" )
      Coil( "E41" )
   END_RUNG
   // the same network as SCL:
   "E41" := NOT "E41";
END_REGION

REGION Network 17: Deceleration for pallet position (Conveyor)
   RUNG wire#powerrail
      I_Contact( "E83" )
      Coil( "E83" )
   END_RUNG
   // the same network as SCL:
   "E83" := NOT "E83";
END_REGION

REGION Network 18: EXCHANGE SIGNALS
END_REGION

REGION Network 19: Pallet ready in infeed signal (Infeed signal)
   RUNG wire#powerrail
      Contact( "E3.6" )
      wire#w1
      Coil( "E121" )
   END_RUNG
   RUNG wire#powerrail
      Contact( "DB22_DisplayData".dbx22_0 )
   END_RUNG wire#w1
   // the same network as SCL:
   "E121" := "E3.6" OR "DB22_DisplayData".dbx22_0;
END_REGION

REGION Network 20: Ready to receive pallet from outfeed signal (Outfeed signal)
   RUNG wire#powerrail
      Contact( "E3.7" )
      wire#w1
      Coil( "E122" )
   END_RUNG
   RUNG wire#powerrail
      Contact( "DB22_DisplayData".dbx22_4 )
   END_RUNG wire#w1
   // the same network as SCL:
   "E122" := "E3.7" OR "DB22_DisplayData".dbx22_4;
END_REGION

REGION Network 21: End of pallet transfer signal (Outfeed signal)
   RUNG wire#powerrail
      Contact( "E4.0" )
      wire#w1
      Coil( "E123" )
   END_RUNG
   RUNG wire#powerrail
      Contact( "DB22_DisplayData".dbx22_5 )
   END_RUNG wire#w1
   // the same network as SCL:
   "E123" := "E4.0" OR "DB22_DisplayData".dbx22_5;
END_REGION

REGION Network 22: Wrapping excluded signal (Std signal)
   RUNG wire#powerrail
      Contact( "E4.1" )
      Coil( "E49" )
   END_RUNG
   // the same network as SCL:
   "E49" := "E4.1";
END_REGION

REGION Network 23: SEGNALE PORTA TAGLIAFUOCO APERTA
   RUNG wire#powerrail
      Contact( "E5.4" )
      Coil( "E117" )
   END_RUNG
   // the same network as SCL:
   "E117" := "E5.4";
END_REGION

REGION Network 24: SEGNALE CHIUSURA PORTA TAGLIAFUOCO
   // RICHIESTA...
   RUNG wire#powerrail
      Contact( "E5.5" )
      Coil( "E118" )
   END_RUNG
   // the same network as SCL:
   "E118" := "E5.5";
END_REGION

REGION Network 25: [B2782] CONTROLLO 1 POSIZIONAMENTO POS. 05
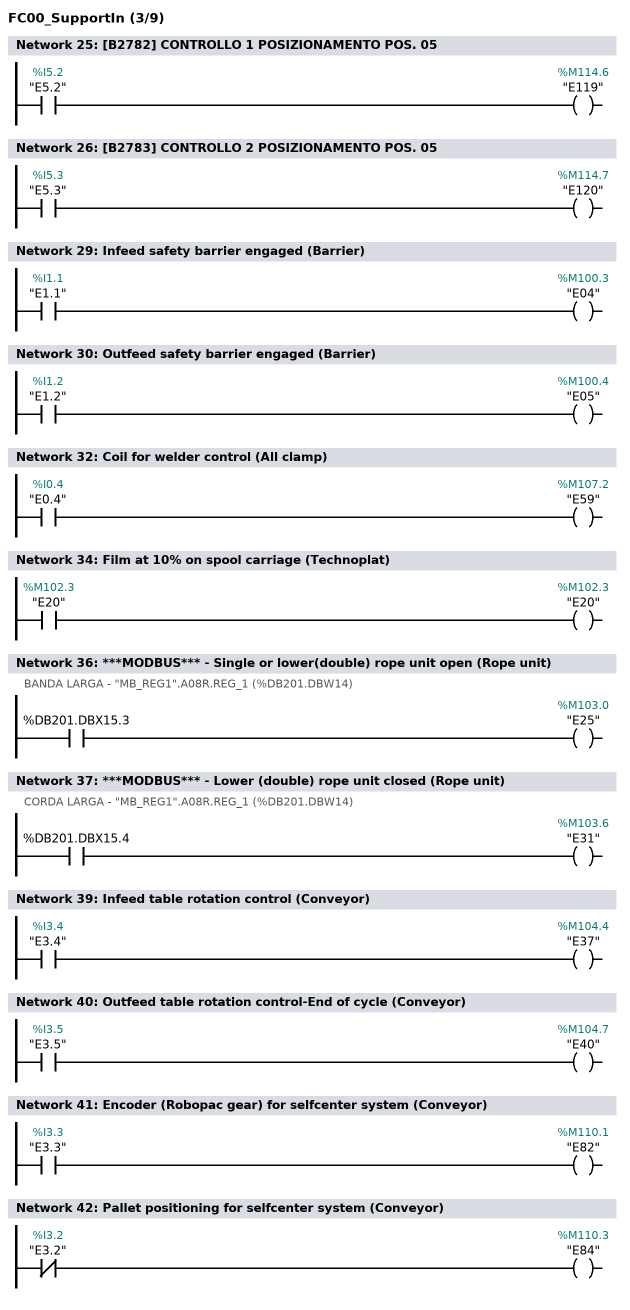
   RUNG wire#powerrail
      Contact( "E5.2" )
      Coil( "E119" )
   END_RUNG
   // the same network as SCL:
   "E119" := "E5.2";
END_REGION

REGION Network 26: [B2783] CONTROLLO 2 POSIZIONAMENTO POS. 05
   RUNG wire#powerrail
      Contact( "E5.3" )
      Coil( "E120" )
   END_RUNG
   // the same network as SCL:
   "E120" := "E5.3";
END_REGION

REGION Network 27: ACCESSORIES
END_REGION

REGION Network 28: ***BARRIERS***
END_REGION

REGION Network 29: Infeed safety barrier engaged (Barrier)
   RUNG wire#powerrail
      Contact( "E1.1" )
      Coil( "E04" )
   END_RUNG
   // the same network as SCL:
   "E04" := "E1.1";
END_REGION

REGION Network 30: Outfeed safety barrier engaged (Barrier)
   RUNG wire#powerrail
      Contact( "E1.2" )
      Coil( "E05" )
   END_RUNG
   // the same network as SCL:
   "E05" := "E1.2";
END_REGION

REGION Network 31: ***WELDER***
END_REGION

REGION Network 32: Coil for welder control (All clamp)
   RUNG wire#powerrail
      Contact( "E0.4" )
      Coil( "E59" )
   END_RUNG
   // the same network as SCL:
   "E59" := "E0.4";
END_REGION

REGION Network 33: ***ES_FILM***
END_REGION

REGION Network 34: Film at 10% on spool carriage (Technoplat)
   RUNG wire#powerrail
      Contact( "E20" )
      Coil( "E20" )
   END_RUNG
   // the same network as SCL:
   "E20" := "E20";
END_REGION

REGION Network 35: ***BAND/ROPE***
END_REGION

REGION Network 36: ***MODBUS*** - Single or lower(double) rope unit open (Rope unit)
   // BANDA LARGA - "MB_REG1".A08R.REG_1 (%DB201.DBW14)
   RUNG wire#powerrail
      Contact( %DB201.DBX15.3 )
      Coil( "E25" )
   END_RUNG
   // the same network as SCL:
   "E25" := %DB201.DBX15.3;
END_REGION

REGION Network 37: ***MODBUS*** - Lower (double) rope unit closed (Rope unit)
   // CORDA LARGA - "MB_REG1".A08R.REG_1 (%DB201.DBW14)
   RUNG wire#powerrail
      Contact( %DB201.DBX15.4 )
      Coil( "E31" )
   END_RUNG
   // the same network as SCL:
   "E31" := %DB201.DBX15.4;
END_REGION

REGION Network 38: ***SELF-CENTER***
END_REGION

REGION Network 39: Infeed table rotation control (Conveyor)
   RUNG wire#powerrail
      Contact( "E3.4" )
      Coil( "E37" )
   END_RUNG
   // the same network as SCL:
   "E37" := "E3.4";
END_REGION

REGION Network 40: Outfeed table rotation control-End of cycle (Conveyor)
   RUNG wire#powerrail
      Contact( "E3.5" )
      Coil( "E40" )
   END_RUNG
   // the same network as SCL:
   "E40" := "E3.5";
END_REGION

REGION Network 41: Encoder (Robopac gear) for selfcenter system (Conveyor)
   RUNG wire#powerrail
      Contact( "E3.3" )
      Coil( "E82" )
   END_RUNG
   // the same network as SCL:
   "E82" := "E3.3";
END_REGION

REGION Network 42: Pallet positioning for selfcenter system (Conveyor)
   RUNG wire#powerrail
      I_Contact( "E3.2" )
      Coil( "E84" )
   END_RUNG
   // the same network as SCL:
   "E84" := NOT "E3.2";
END_REGION

REGION Network 43: ***CONTRAST***
END_REGION

REGION Network 44: Welder contrast back (Contrast carriage)
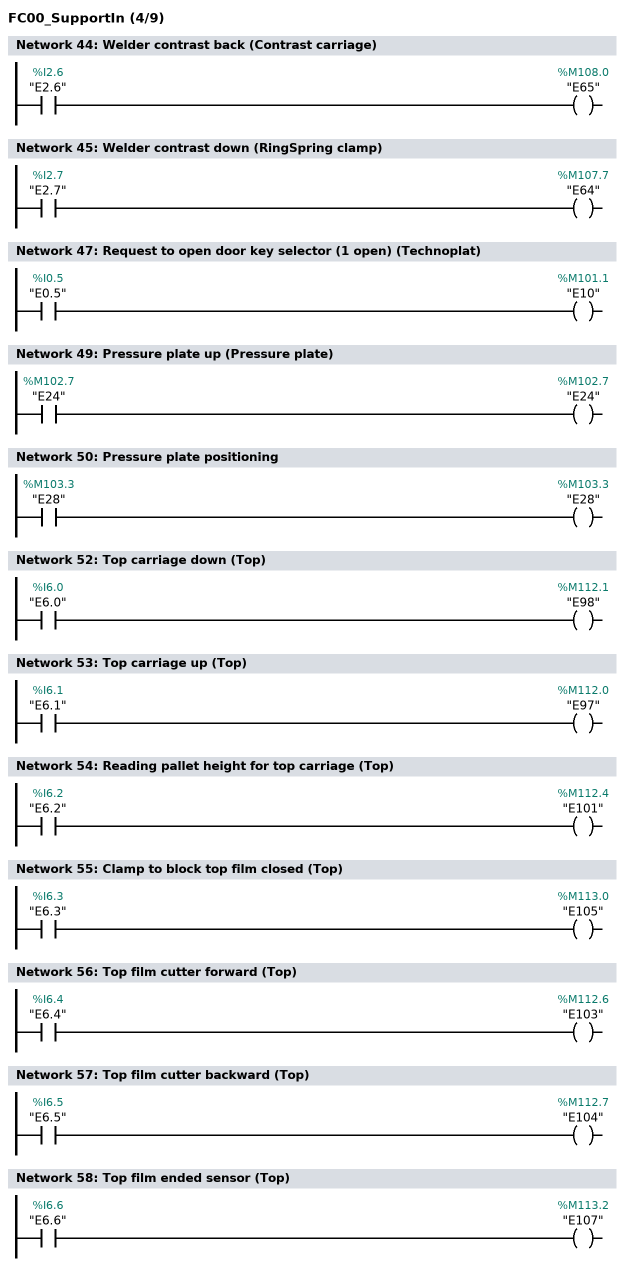
   RUNG wire#powerrail
      Contact( "E2.6" )
      Coil( "E65" )
   END_RUNG
   // the same network as SCL:
   "E65" := "E2.6";
END_REGION

REGION Network 45: Welder contrast down (RingSpring clamp)
   RUNG wire#powerrail
      Contact( "E2.7" )
      Coil( "E64" )
   END_RUNG
   // the same network as SCL:
   "E64" := "E2.7";
END_REGION

REGION Network 46: ***DOOR***
END_REGION

REGION Network 47: Request to open door key selector (1 open) (Technoplat)
   RUNG wire#powerrail
      Contact( "E0.5" )
      Coil( "E10" )
   END_RUNG
   // the same network as SCL:
   "E10" := "E0.5";
END_REGION

REGION Network 48: ***PRESSURE***
END_REGION

REGION Network 49: Pressure plate up (Pressure plate)
   RUNG wire#powerrail
      Contact( "E24" )
      Coil( "E24" )
   END_RUNG
   // the same network as SCL:
   "E24" := "E24";
END_REGION

REGION Network 50: Pressure plate positioning
   RUNG wire#powerrail
      Contact( "E28" )
      Coil( "E28" )
   END_RUNG
   // the same network as SCL:
   "E28" := "E28";
END_REGION

REGION Network 51: ***TOP***
END_REGION

REGION Network 52: Top carriage down (Top)
   RUNG wire#powerrail
      Contact( "E6.0" )
      Coil( "E98" )
   END_RUNG
   // the same network as SCL:
   "E98" := "E6.0";
END_REGION

REGION Network 53: Top carriage up (Top)
   RUNG wire#powerrail
      Contact( "E6.1" )
      Coil( "E97" )
   END_RUNG
   // the same network as SCL:
   "E97" := "E6.1";
END_REGION

REGION Network 54: Reading pallet height for top carriage (Top)
   RUNG wire#powerrail
      Contact( "E6.2" )
      Coil( "E101" )
   END_RUNG
   // the same network as SCL:
   "E101" := "E6.2";
END_REGION

REGION Network 55: Clamp to block top film closed (Top)
   RUNG wire#powerrail
      Contact( "E6.3" )
      Coil( "E105" )
   END_RUNG
   // the same network as SCL:
   "E105" := "E6.3";
END_REGION

REGION Network 56: Top film cutter forward (Top)
   RUNG wire#powerrail
      Contact( "E6.4" )
      Coil( "E103" )
   END_RUNG
   // the same network as SCL:
   "E103" := "E6.4";
END_REGION

REGION Network 57: Top film cutter backward (Top)
   RUNG wire#powerrail
      Contact( "E6.5" )
      Coil( "E104" )
   END_RUNG
   // the same network as SCL:
   "E104" := "E6.5";
END_REGION

REGION Network 58: Top film ended sensor (Top)
   RUNG wire#powerrail
      Contact( "E6.6" )
      Coil( "E107" )
   END_RUNG
   // the same network as SCL:
   "E107" := "E6.6";
END_REGION

REGION Network 59: Top carriage position under pressure plate (Top)
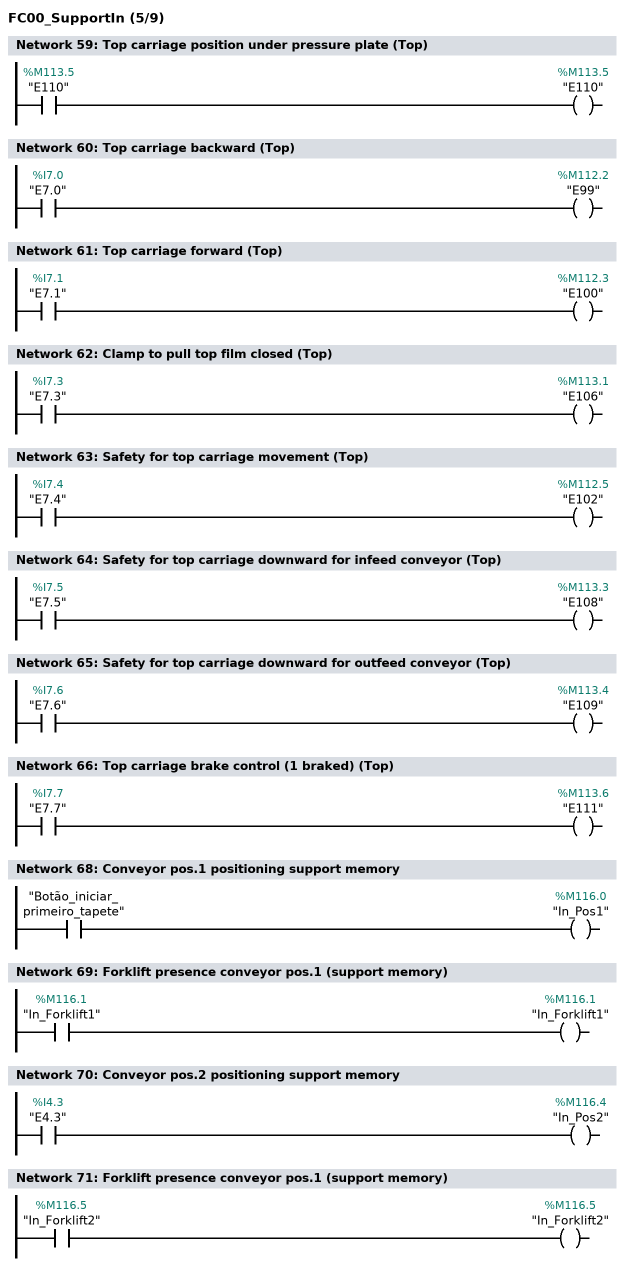
   RUNG wire#powerrail
      Contact( "E110" )
      Coil( "E110" )
   END_RUNG
   // the same network as SCL:
   "E110" := "E110";
END_REGION

REGION Network 60: Top carriage backward (Top)
   RUNG wire#powerrail
      Contact( "E7.0" )
      Coil( "E99" )
   END_RUNG
   // the same network as SCL:
   "E99" := "E7.0";
END_REGION

REGION Network 61: Top carriage forward (Top)
   RUNG wire#powerrail
      Contact( "E7.1" )
      Coil( "E100" )
   END_RUNG
   // the same network as SCL:
   "E100" := "E7.1";
END_REGION

REGION Network 62: Clamp to pull top film closed (Top)
   RUNG wire#powerrail
      Contact( "E7.3" )
      Coil( "E106" )
   END_RUNG
   // the same network as SCL:
   "E106" := "E7.3";
END_REGION

REGION Network 63: Safety for top carriage movement (Top)
   RUNG wire#powerrail
      Contact( "E7.4" )
      Coil( "E102" )
   END_RUNG
   // the same network as SCL:
   "E102" := "E7.4";
END_REGION

REGION Network 64: Safety for top carriage downward for infeed conveyor (Top)
   RUNG wire#powerrail
      Contact( "E7.5" )
      Coil( "E108" )
   END_RUNG
   // the same network as SCL:
   "E108" := "E7.5";
END_REGION

REGION Network 65: Safety for top carriage downward for outfeed conveyor (Top)
   RUNG wire#powerrail
      Contact( "E7.6" )
      Coil( "E109" )
   END_RUNG
   // the same network as SCL:
   "E109" := "E7.6";
END_REGION

REGION Network 66: Top carriage brake control (1 braked) (Top)
   RUNG wire#powerrail
      Contact( "E7.7" )
      Coil( "E111" )
   END_RUNG
   // the same network as SCL:
   "E111" := "E7.7";
END_REGION

REGION Network 67: ***CONVEYORS***
END_REGION

REGION Network 68: Conveyor pos.1 positioning support memory
   RUNG wire#powerrail
      Contact( "Botão_iniciar_primeiro_tapete" )
      Coil( "In_Pos1" )
   END_RUNG
   // the same network as SCL:
   "In_Pos1" := "Botão_iniciar_primeiro_tapete";
END_REGION

REGION Network 69: Forklift presence conveyor pos.1 (support memory)
   RUNG wire#powerrail
      Contact( "In_Forklift1" )
      Coil( "In_Forklift1" )
   END_RUNG
   // the same network as SCL:
   "In_Forklift1" := "In_Forklift1";
END_REGION

REGION Network 70: Conveyor pos.2 positioning support memory
   RUNG wire#powerrail
      Contact( "E4.3" )
      Coil( "In_Pos2" )
   END_RUNG
   // the same network as SCL:
   "In_Pos2" := "E4.3";
END_REGION

REGION Network 71: Forklift presence conveyor pos.1 (support memory)
   RUNG wire#powerrail
      Contact( "In_Forklift2" )
      Coil( "In_Forklift2" )
   END_RUNG
   // the same network as SCL:
   "In_Forklift2" := "In_Forklift2";
END_REGION

REGION Network 72: Conveyor pos.3 positioning support memory
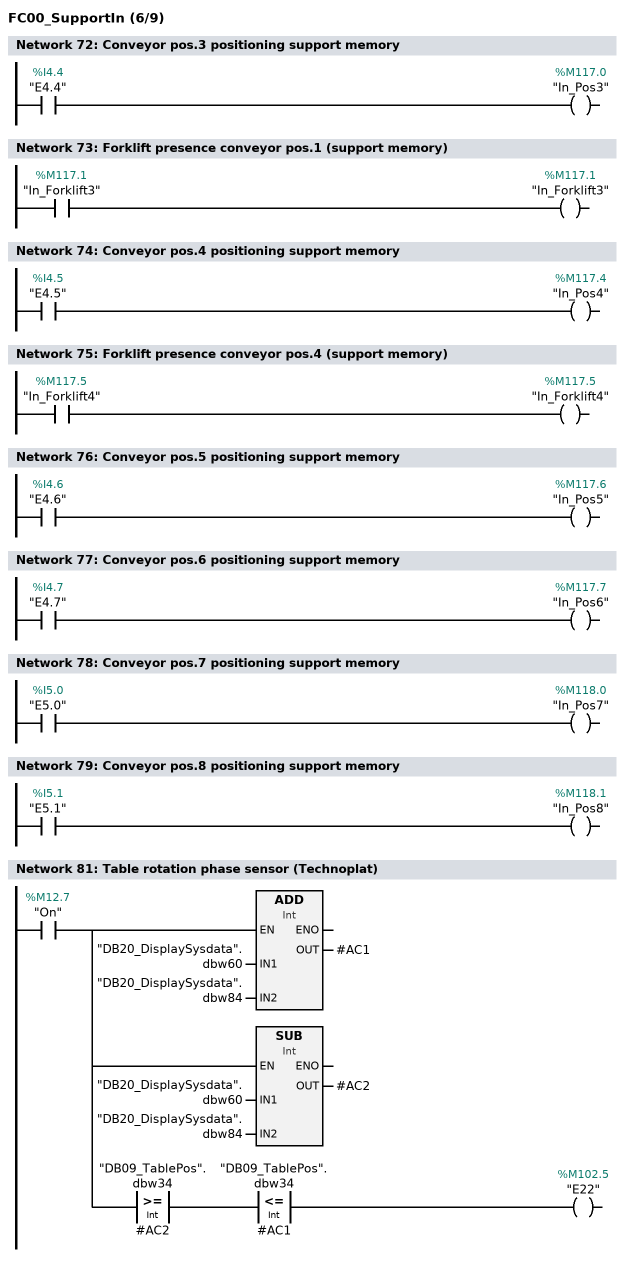
   RUNG wire#powerrail
      Contact( "E4.4" )
      Coil( "In_Pos3" )
   END_RUNG
   // the same network as SCL:
   "In_Pos3" := "E4.4";
END_REGION

REGION Network 73: Forklift presence conveyor pos.1 (support memory)
   RUNG wire#powerrail
      Contact( "In_Forklift3" )
      Coil( "In_Forklift3" )
   END_RUNG
   // the same network as SCL:
   "In_Forklift3" := "In_Forklift3";
END_REGION

REGION Network 74: Conveyor pos.4 positioning support memory
   RUNG wire#powerrail
      Contact( "E4.5" )
      Coil( "In_Pos4" )
   END_RUNG
   // the same network as SCL:
   "In_Pos4" := "E4.5";
END_REGION

REGION Network 75: Forklift presence conveyor pos.4 (support memory)
   RUNG wire#powerrail
      Contact( "In_Forklift4" )
      Coil( "In_Forklift4" )
   END_RUNG
   // the same network as SCL:
   "In_Forklift4" := "In_Forklift4";
END_REGION

REGION Network 76: Conveyor pos.5 positioning support memory
   RUNG wire#powerrail
      Contact( "E4.6" )
      Coil( "In_Pos5" )
   END_RUNG
   // the same network as SCL:
   "In_Pos5" := "E4.6";
END_REGION

REGION Network 77: Conveyor pos.6 positioning support memory
   RUNG wire#powerrail
      Contact( "E4.7" )
      Coil( "In_Pos6" )
   END_RUNG
   // the same network as SCL:
   "In_Pos6" := "E4.7";
END_REGION

REGION Network 78: Conveyor pos.7 positioning support memory
   RUNG wire#powerrail
      Contact( "E5.0" )
      Coil( "In_Pos7" )
   END_RUNG
   // the same network as SCL:
   "In_Pos7" := "E5.0";
END_REGION

REGION Network 79: Conveyor pos.8 positioning support memory
   RUNG wire#powerrail
      Contact( "E5.1" )
      Coil( "In_Pos8" )
   END_RUNG
   // the same network as SCL:
   "In_Pos8" := "E5.1";
END_REGION

REGION Network 80: OTHER
END_REGION

REGION Network 81: Table rotation phase sensor (Technoplat)
   RUNG wire#powerrail
      Contact( "On" )
      wire#w1
      { S7_Templates := "SrcType := Int"; S7_GenerateENO := "TRUE" } Add(in1 := "DB20_DisplaySysdata".dbw60, in2 := "DB20_DisplaySysdata".dbw84, out => #AC1)
   END_RUNG
   RUNG wire#w1
      { S7_Templates := "SrcType := Int"; S7_GenerateENO := "TRUE" } Sub(in1 := "DB20_DisplaySysdata".dbw60, in2 := "DB20_DisplaySysdata".dbw84, out => #AC2)
   END_RUNG
   RUNG wire#w1
      { S7_Templates := "SrcType := Int" } GE_Contact(in1 := "DB09_TablePos".dbw34, in2 := #AC2)
      { S7_Templates := "SrcType := Int" } LE_Contact(in1 := "DB09_TablePos".dbw34, in2 := #AC1)
      Coil( "E22" )
   END_RUNG
   // the same network as SCL:
   IF "On" THEN
       #AC1 := "DB20_DisplaySysdata".dbw60 + "DB20_DisplaySysdata".dbw84;
       #AC2 := "DB20_DisplaySysdata".dbw60 - "DB20_DisplaySysdata".dbw84;
   END_IF;
   "E22" := "On" AND ("DB09_TablePos".dbw34 >= #AC2) AND ("DB09_TablePos".dbw34 <= #AC1);
END_REGION

REGION Network 82: Table rotation load phase sensor (Technoplat)
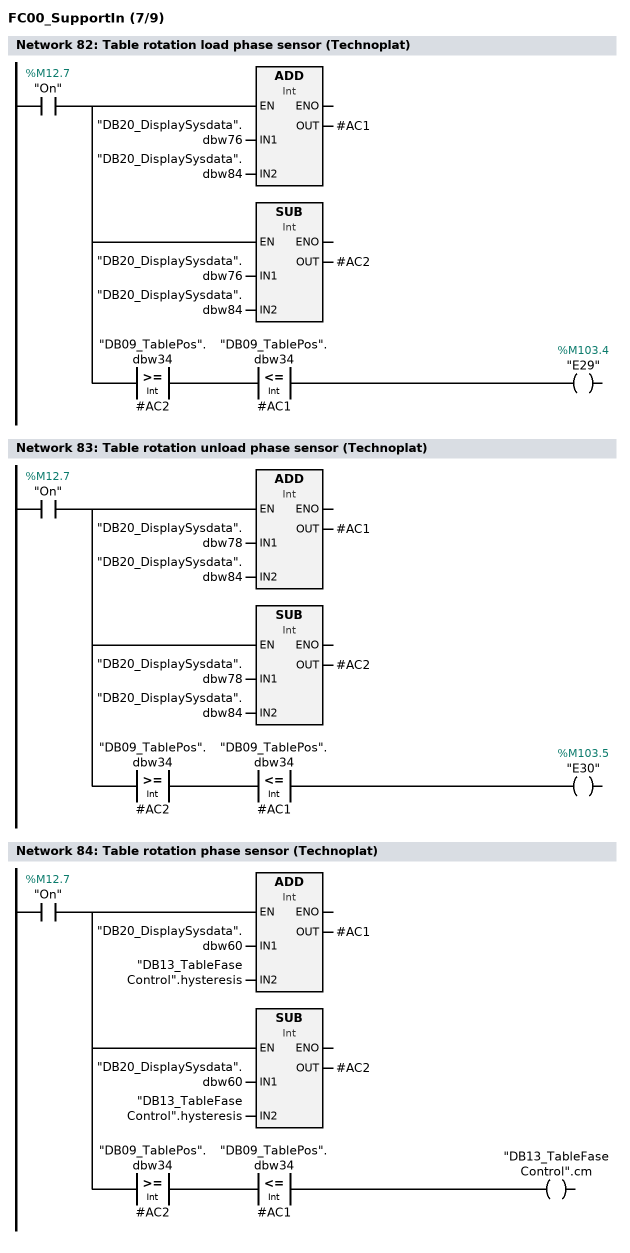
   RUNG wire#powerrail
      Contact( "On" )
      wire#w1
      { S7_Templates := "SrcType := Int"; S7_GenerateENO := "TRUE" } Add(in1 := "DB20_DisplaySysdata".dbw76, in2 := "DB20_DisplaySysdata".dbw84, out => #AC1)
   END_RUNG
   RUNG wire#w1
      { S7_Templates := "SrcType := Int"; S7_GenerateENO := "TRUE" } Sub(in1 := "DB20_DisplaySysdata".dbw76, in2 := "DB20_DisplaySysdata".dbw84, out => #AC2)
   END_RUNG
   RUNG wire#w1
      { S7_Templates := "SrcType := Int" } GE_Contact(in1 := "DB09_TablePos".dbw34, in2 := #AC2)
      { S7_Templates := "SrcType := Int" } LE_Contact(in1 := "DB09_TablePos".dbw34, in2 := #AC1)
      Coil( "E29" )
   END_RUNG
   // the same network as SCL:
   IF "On" THEN
       #AC1 := "DB20_DisplaySysdata".dbw76 + "DB20_DisplaySysdata".dbw84;
       #AC2 := "DB20_DisplaySysdata".dbw76 - "DB20_DisplaySysdata".dbw84;
   END_IF;
   "E29" := "On" AND ("DB09_TablePos".dbw34 >= #AC2) AND ("DB09_TablePos".dbw34 <= #AC1);
END_REGION

REGION Network 83: Table rotation unload phase sensor (Technoplat)
   RUNG wire#powerrail
      Contact( "On" )
      wire#w1
      { S7_Templates := "SrcType := Int"; S7_GenerateENO := "TRUE" } Add(in1 := "DB20_DisplaySysdata".dbw78, in2 := "DB20_DisplaySysdata".dbw84, out => #AC1)
   END_RUNG
   RUNG wire#w1
      { S7_Templates := "SrcType := Int"; S7_GenerateENO := "TRUE" } Sub(in1 := "DB20_DisplaySysdata".dbw78, in2 := "DB20_DisplaySysdata".dbw84, out => #AC2)
   END_RUNG
   RUNG wire#w1
      { S7_Templates := "SrcType := Int" } GE_Contact(in1 := "DB09_TablePos".dbw34, in2 := #AC2)
      { S7_Templates := "SrcType := Int" } LE_Contact(in1 := "DB09_TablePos".dbw34, in2 := #AC1)
      Coil( "E30" )
   END_RUNG
   // the same network as SCL:
   IF "On" THEN
       #AC1 := "DB20_DisplaySysdata".dbw78 + "DB20_DisplaySysdata".dbw84;
       #AC2 := "DB20_DisplaySysdata".dbw78 - "DB20_DisplaySysdata".dbw84;
   END_IF;
   "E30" := "On" AND ("DB09_TablePos".dbw34 >= #AC2) AND ("DB09_TablePos".dbw34 <= #AC1);
END_REGION

REGION Network 84: Table rotation phase sensor (Technoplat)
   RUNG wire#powerrail
      Contact( "On" )
      wire#w1
      { S7_Templates := "SrcType := Int"; S7_GenerateENO := "TRUE" } Add(in1 := "DB20_DisplaySysdata".dbw60, in2 := "DB13_TableFaseControl".hysteresis, out => #AC1)
   END_RUNG
   RUNG wire#w1
      { S7_Templates := "SrcType := Int"; S7_GenerateENO := "TRUE" } Sub(in1 := "DB20_DisplaySysdata".dbw60, in2 := "DB13_TableFaseControl".hysteresis, out => #AC2)
   END_RUNG
   RUNG wire#w1
      { S7_Templates := "SrcType := Int" } GE_Contact(in1 := "DB09_TablePos".dbw34, in2 := #AC2)
      { S7_Templates := "SrcType := Int" } LE_Contact(in1 := "DB09_TablePos".dbw34, in2 := #AC1)
      Coil( "DB13_TableFaseControl".cm )
   END_RUNG
   // the same network as SCL:
   IF "On" THEN
       #AC1 := "DB20_DisplaySysdata".dbw60 + "DB13_TableFaseControl".hysteresis;
       #AC2 := "DB20_DisplaySysdata".dbw60 - "DB13_TableFaseControl".hysteresis;
   END_IF;
   "DB13_TableFaseControl".cm := "On" AND ("DB09_TablePos".dbw34 >= #AC2) AND ("DB09_TablePos".dbw34 <= #AC1);
END_REGION

REGION Network 85: Table rotation load phase sensor (Technoplat)
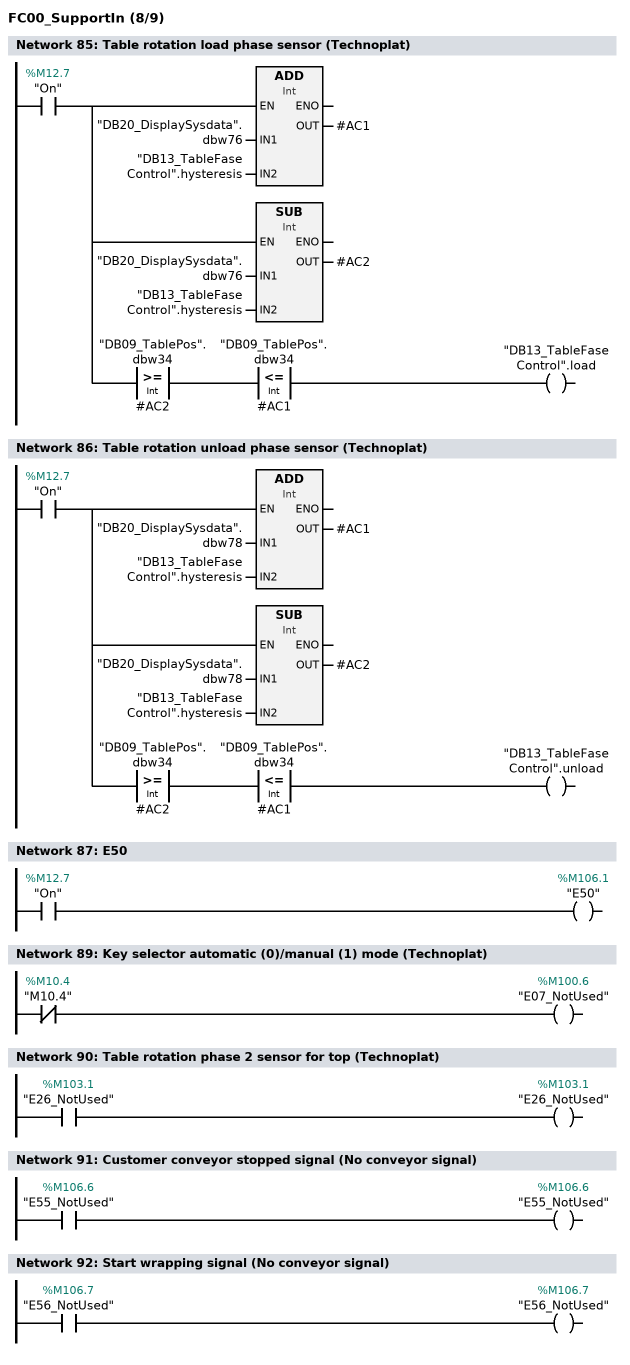
   RUNG wire#powerrail
      Contact( "On" )
      wire#w1
      { S7_Templates := "SrcType := Int"; S7_GenerateENO := "TRUE" } Add(in1 := "DB20_DisplaySysdata".dbw76, in2 := "DB13_TableFaseControl".hysteresis, out => #AC1)
   END_RUNG
   RUNG wire#w1
      { S7_Templates := "SrcType := Int"; S7_GenerateENO := "TRUE" } Sub(in1 := "DB20_DisplaySysdata".dbw76, in2 := "DB13_TableFaseControl".hysteresis, out => #AC2)
   END_RUNG
   RUNG wire#w1
      { S7_Templates := "SrcType := Int" } GE_Contact(in1 := "DB09_TablePos".dbw34, in2 := #AC2)
      { S7_Templates := "SrcType := Int" } LE_Contact(in1 := "DB09_TablePos".dbw34, in2 := #AC1)
      Coil( "DB13_TableFaseControl".load )
   END_RUNG
   // the same network as SCL:
   IF "On" THEN
       #AC1 := "DB20_DisplaySysdata".dbw76 + "DB13_TableFaseControl".hysteresis;
       #AC2 := "DB20_DisplaySysdata".dbw76 - "DB13_TableFaseControl".hysteresis;
   END_IF;
   "DB13_TableFaseControl".load := "On" AND ("DB09_TablePos".dbw34 >= #AC2) AND ("DB09_TablePos".dbw34 <= #AC1);
END_REGION

REGION Network 86: Table rotation unload phase sensor (Technoplat)
   RUNG wire#powerrail
      Contact( "On" )
      wire#w1
      { S7_Templates := "SrcType := Int"; S7_GenerateENO := "TRUE" } Add(in1 := "DB20_DisplaySysdata".dbw78, in2 := "DB13_TableFaseControl".hysteresis, out => #AC1)
   END_RUNG
   RUNG wire#w1
      { S7_Templates := "SrcType := Int"; S7_GenerateENO := "TRUE" } Sub(in1 := "DB20_DisplaySysdata".dbw78, in2 := "DB13_TableFaseControl".hysteresis, out => #AC2)
   END_RUNG
   RUNG wire#w1
      { S7_Templates := "SrcType := Int" } GE_Contact(in1 := "DB09_TablePos".dbw34, in2 := #AC2)
      { S7_Templates := "SrcType := Int" } LE_Contact(in1 := "DB09_TablePos".dbw34, in2 := #AC1)
      Coil( "DB13_TableFaseControl".unload )
   END_RUNG
   // the same network as SCL:
   IF "On" THEN
       #AC1 := "DB20_DisplaySysdata".dbw78 + "DB13_TableFaseControl".hysteresis;
       #AC2 := "DB20_DisplaySysdata".dbw78 - "DB13_TableFaseControl".hysteresis;
   END_IF;
   "DB13_TableFaseControl".unload := "On" AND ("DB09_TablePos".dbw34 >= #AC2) AND ("DB09_TablePos".dbw34 <= #AC1);
END_REGION

REGION Network 87: E50
   RUNG wire#powerrail
      Contact( "On" )
      Coil( "E50" )
   END_RUNG
   // the same network as SCL:
   "E50" := "On";
END_REGION

REGION Network 88: OLD (NOT USED)
END_REGION

REGION Network 89: Key selector automatic (0)/manual (1) mode (Technoplat)
   RUNG wire#powerrail
      I_Contact( "M10.4" )
      Coil( "E07_NotUsed" )
   END_RUNG
   // the same network as SCL:
   "E07_NotUsed" := NOT "M10.4";
END_REGION

REGION Network 90: Table rotation phase 2 sensor for top (Technoplat)
   RUNG wire#powerrail
      Contact( "E26_NotUsed" )
      Coil( "E26_NotUsed" )
   END_RUNG
   // the same network as SCL:
   "E26_NotUsed" := "E26_NotUsed";
END_REGION

REGION Network 91: Customer conveyor stopped signal (No conveyor signal)
   RUNG wire#powerrail
      Contact( "E55_NotUsed" )
      Coil( "E55_NotUsed" )
   END_RUNG
   // the same network as SCL:
   "E55_NotUsed" := "E55_NotUsed";
END_REGION

REGION Network 92: Start wrapping signal (No conveyor signal)
   RUNG wire#powerrail
      Contact( "E56_NotUsed" )
      Coil( "E56_NotUsed" )
   END_RUNG
   // the same network as SCL:
   "E56_NotUsed" := "E56_NotUsed";
END_REGION

REGION Network 93: Film clamp down (RingSpring clamp)
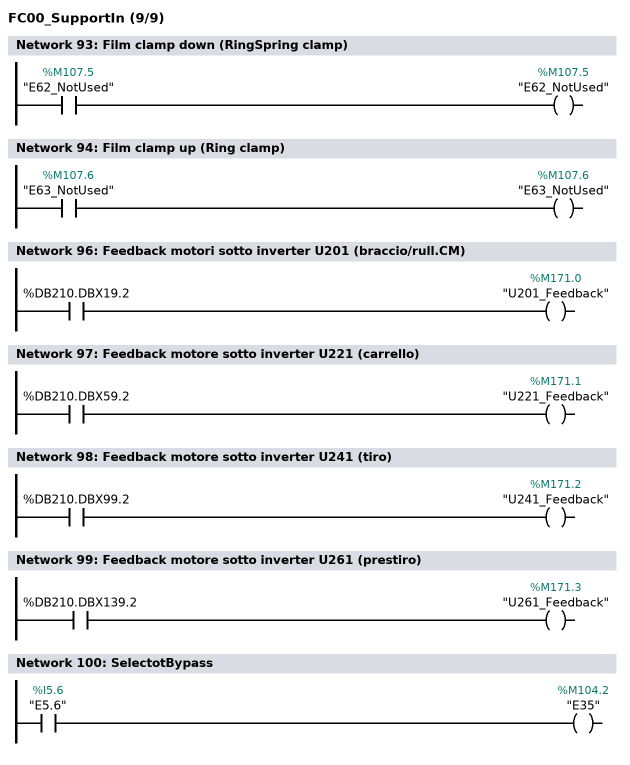
   RUNG wire#powerrail
      Contact( "E62_NotUsed" )
      Coil( "E62_NotUsed" )
   END_RUNG
   // the same network as SCL:
   "E62_NotUsed" := "E62_NotUsed";
END_REGION

REGION Network 94: Film clamp up (Ring clamp)
   RUNG wire#powerrail
      Contact( "E63_NotUsed" )
      Coil( "E63_NotUsed" )
   END_RUNG
   // the same network as SCL:
   "E63_NotUsed" := "E63_NotUsed";
END_REGION

REGION Network 95: PROFINET DATA (inverter)
END_REGION

REGION Network 96: Feedback motori sotto inverter U201 (braccio/rull.CM)
   RUNG wire#powerrail
      Contact( %DB210.DBX19.2 )
      Coil( "U201_Feedback" )
   END_RUNG
   // the same network as SCL:
   "U201_Feedback" := %DB210.DBX19.2;
END_REGION

REGION Network 97: Feedback motore sotto inverter U221 (carrello)
   RUNG wire#powerrail
      Contact( %DB210.DBX59.2 )
      Coil( "U221_Feedback" )
   END_RUNG
   // the same network as SCL:
   "U221_Feedback" := %DB210.DBX59.2;
END_REGION

REGION Network 98: Feedback motore sotto inverter U241 (tiro)
   RUNG wire#powerrail
      Contact( %DB210.DBX99.2 )
      Coil( "U241_Feedback" )
   END_RUNG
   // the same network as SCL:
   "U241_Feedback" := %DB210.DBX99.2;
END_REGION

REGION Network 99: Feedback motore sotto inverter U261 (prestiro)
   RUNG wire#powerrail
      Contact( %DB210.DBX139.2 )
      Coil( "U261_Feedback" )
   END_RUNG
   // the same network as SCL:
   "U261_Feedback" := %DB210.DBX139.2;
END_REGION

REGION Network 100: SelectotBypass
   RUNG wire#powerrail
      Contact( "E5.6" )
      Coil( "E35" )
   END_RUNG
   // the same network as SCL:
   "E35" := "E5.6";
END_REGION
END_FUNCTION

FUNCTION "FC02_Technoplat_TandC" : Void   // FC2, LAD
TITLE = Technoplat timer and counter
{ S7_Optimized_Access := 'FALSE' }
AUTHOR : Robopac
VERSION : 0.0
// stored: AutoNumber false, IsIECCheckEnabled false, SetENOAutomatically false, UDAEnableTagReadback false
   VAR_INPUT
      FASTSPEED : Bool;
   END_VAR
   VAR_TEMP
      TempInt : Int;
      TempDint : DInt;
   END_VAR
   VAR_TEMP   // added for the SCL form of the ladder/FBD networks
      _w1 : Bool;
      _w2 : Bool;
   END_VAR
BEGIN

REGION Network 1: Time to filter inverter alarms
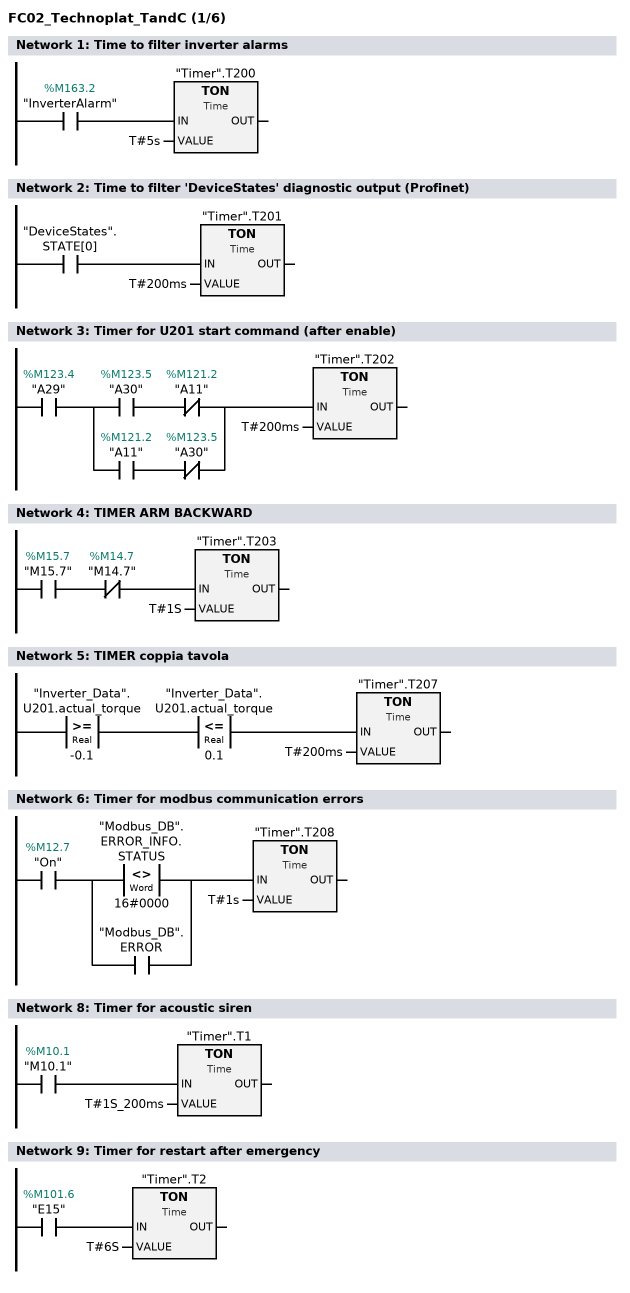
   "Timer".T200.TON(IN := "InverterAlarm", PT := T#5s);   // TON coil
END_REGION

REGION Network 2: Time to filter 'DeviceStates' diagnostic output (Profinet)
   "Timer".T201.TON(IN := "DeviceStates".STATE[0], PT := T#200ms);   // TON coil
END_REGION

REGION Network 3: Timer for U201 start command (after enable)
   "Timer".T202.TON(IN := "A29" AND (("A30" AND NOT "A11") OR ("A11" AND NOT "A30")), PT := T#200ms);   // TON coil
END_REGION

REGION Network 4: TIMER ARM BACKWARD
   "Timer".T203.TON(IN := "M15.7" AND NOT "M14.7", PT := T#1S);   // TON coil
END_REGION

REGION Network 5: TIMER coppia tavola
   "Timer".T207.TON(IN := ("Inverter_Data".U201.actual_torque >= (-0.1)) AND ("Inverter_Data".U201.actual_torque <= 0.1), PT := T#200ms);   // TON coil
END_REGION

REGION Network 6: Timer for modbus communication errors
   "Timer".T208.TON(IN := "On" AND (("Modbus_DB".ERROR_INFO.STATUS <> 16#0000) OR "Modbus_DB".ERROR), PT := T#1s);   // TON coil
END_REGION

REGION Network 7: TECHNOPLAT3000
END_REGION

REGION Network 8: Timer for acoustic siren
   "Timer".T1.TON(IN := "M10.1", PT := T#1S_200ms);   // TON coil
END_REGION

REGION Network 9: Timer for restart after emergency
   "Timer".T2.TON(IN := "E15", PT := T#6S);   // TON coil
END_REGION

REGION Network 10: Timer to reset emergency
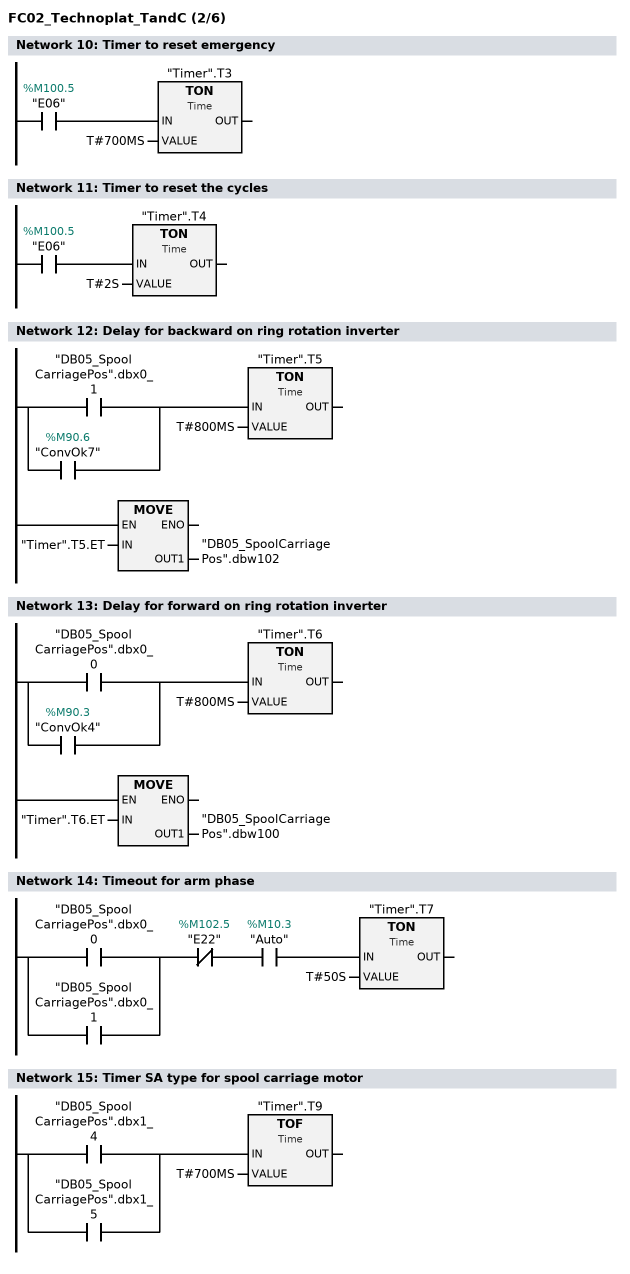
   "Timer".T3.TON(IN := "E06", PT := T#700MS);   // TON coil
END_REGION

REGION Network 11: Timer to reset the cycles
   "Timer".T4.TON(IN := "E06", PT := T#2S);   // TON coil
END_REGION

REGION Network 12: Delay for backward on ring rotation inverter
   "Timer".T5.TON(IN := "DB05_SpoolCarriagePos".dbx0_1 OR "ConvOk7", PT := T#800MS);   // TON coil
   "DB05_SpoolCarriagePos".dbw102 := "Timer".T5.ET;
END_REGION

REGION Network 13: Delay for forward on ring rotation inverter
   "Timer".T6.TON(IN := "DB05_SpoolCarriagePos".dbx0_0 OR "ConvOk4", PT := T#800MS);   // TON coil
   "DB05_SpoolCarriagePos".dbw100 := "Timer".T6.ET;
END_REGION

REGION Network 14: Timeout for arm phase
   "Timer".T7.TON(IN := ("DB05_SpoolCarriagePos".dbx0_0 OR "DB05_SpoolCarriagePos".dbx0_1) AND NOT "E22" AND "Auto", PT := T#50S);   // TON coil
END_REGION

REGION Network 15: Timer SA type for spool carriage motor
   "Timer".T9.TOF(IN := "DB05_SpoolCarriagePos".dbx1_4 OR "DB05_SpoolCarriagePos".dbx1_5, PT := T#700MS);   // TOF coil
END_REGION

REGION Network 16: Timer SA type for arm rotation motor
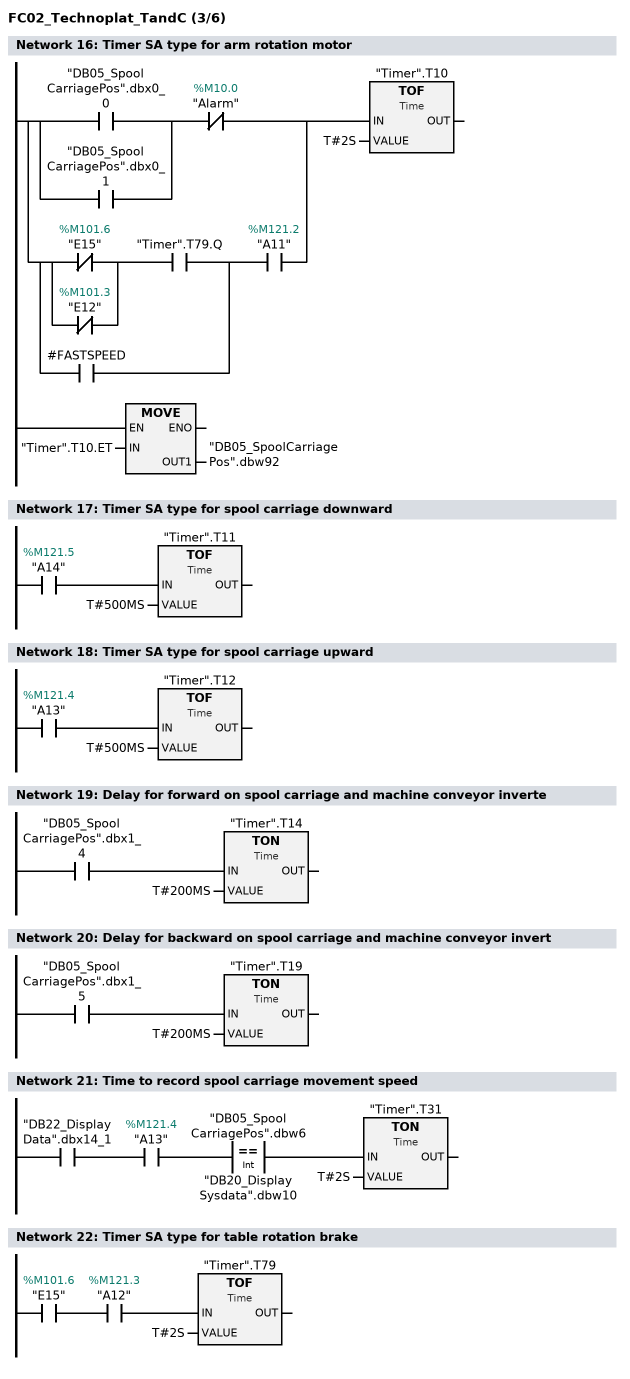
   "Timer".T10.TOF(IN := (("DB05_SpoolCarriagePos".dbx0_0 OR "DB05_SpoolCarriagePos".dbx0_1) AND NOT "Alarm") OR ((((NOT "E15" OR NOT "E12") AND "Timer".T79.Q) OR #FASTSPEED) AND "A11"), PT := T#2S);   // TOF coil
   "DB05_SpoolCarriagePos".dbw92 := "Timer".T10.ET;
END_REGION

REGION Network 17: Timer SA type for spool carriage downward
   "Timer".T11.TOF(IN := "A14", PT := T#500MS);   // TOF coil
END_REGION

REGION Network 18: Timer SA type for spool carriage upward
   "Timer".T12.TOF(IN := "A13", PT := T#500MS);   // TOF coil
END_REGION

REGION Network 19: Delay for forward on spool carriage and machine conveyor inverte
   "Timer".T14.TON(IN := "DB05_SpoolCarriagePos".dbx1_4, PT := T#200MS);   // TON coil
END_REGION

REGION Network 20: Delay for backward on spool carriage and machine conveyor invert
   "Timer".T19.TON(IN := "DB05_SpoolCarriagePos".dbx1_5, PT := T#200MS);   // TON coil
END_REGION

REGION Network 21: Time to record spool carriage movement speed
   "Timer".T31.TON(IN := "DB22_DisplayData".dbx14_1 AND "A13" AND ("DB05_SpoolCarriagePos".dbw6 = "DB20_DisplaySysdata".dbw10), PT := T#2S);   // TON coil
END_REGION

REGION Network 22: Timer SA type for table rotation brake
   "Timer".T79.TOF(IN := "E15" AND "A12", PT := T#2S);   // TOF coil
END_REGION

REGION Network 23: T87: Timer for slow conveyor manual movement
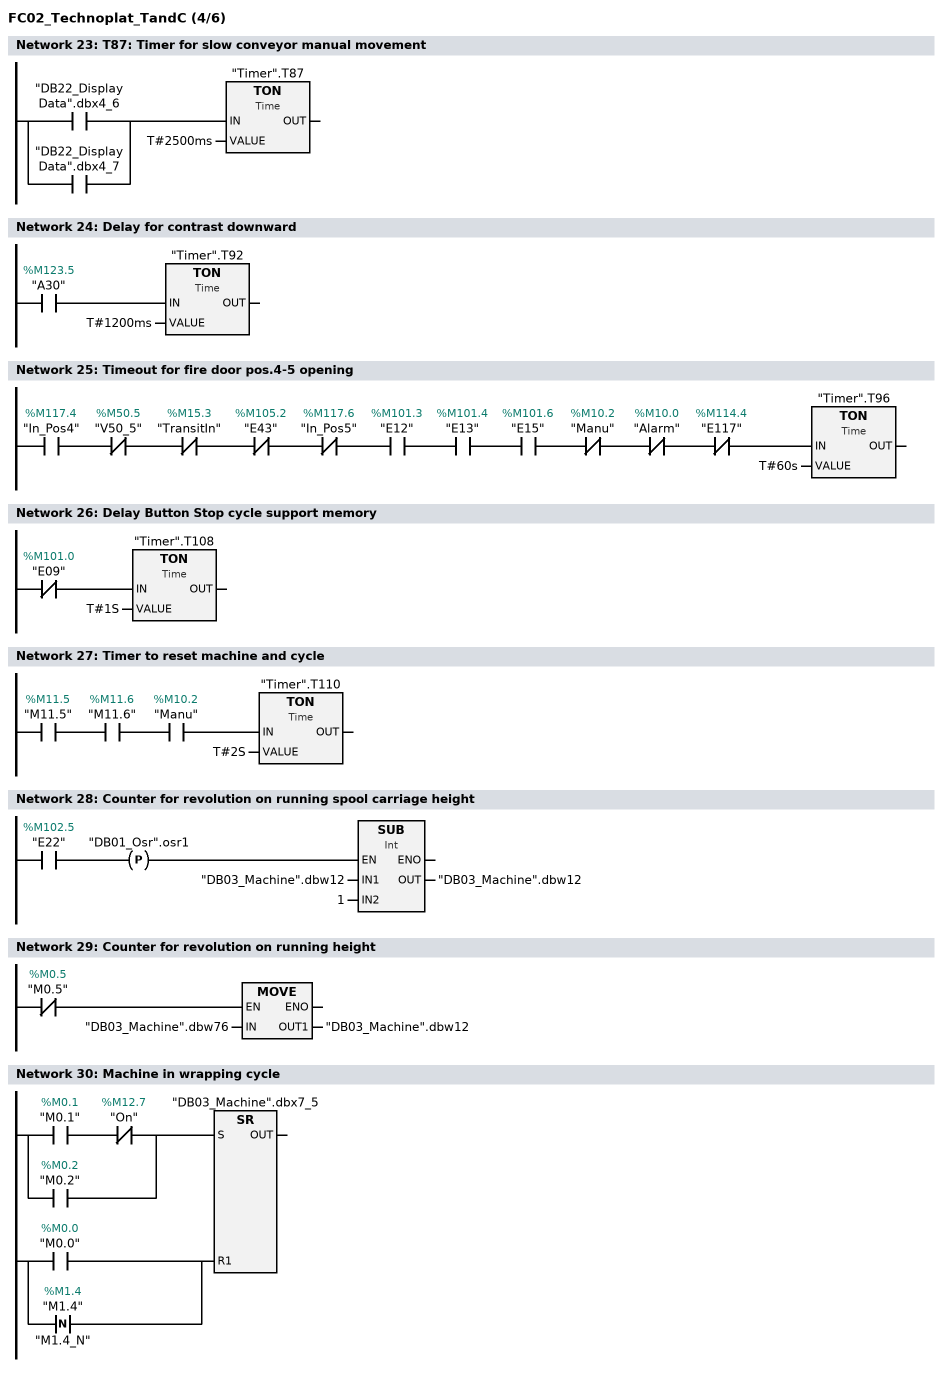
   "Timer".T87.TON(IN := "DB22_DisplayData".dbx4_6 OR "DB22_DisplayData".dbx4_7, PT := T#2500ms);   // TON coil
END_REGION

REGION Network 24: Delay for contrast downward
   "Timer".T92.TON(IN := "A30", PT := T#1200ms);   // TON coil
END_REGION

REGION Network 25: Timeout for fire door pos.4-5 opening
   "Timer".T96.TON(IN := "In_Pos4" AND NOT "V50_5" AND NOT "TransitIn" AND NOT "E43" AND NOT "In_Pos5" AND "E12" AND "E13" AND "E15" AND NOT "Manu" AND NOT "Alarm" AND NOT "E117", PT := T#60s);   // TON coil
END_REGION

REGION Network 26: Delay Button Stop cycle support memory
   "Timer".T108.TON(IN := NOT "E09", PT := T#1S);   // TON coil
END_REGION

REGION Network 27: Timer to reset machine and cycle
   "Timer".T110.TON(IN := "M11.5" AND "M11.6" AND "Manu", PT := T#2S);   // TON coil
END_REGION

REGION Network 28: Counter for revolution on running spool carriage height
   RUNG wire#powerrail
      Contact( "E22" )
      P_Trig( "DB01_Osr".osr1 )
      { S7_Templates := "SrcType := Int"; S7_GenerateENO := "TRUE" } Sub(in1 := "DB03_Machine".dbw12, in2 := 1, out => "DB03_Machine".dbw12)
   END_RUNG
   // the same network as SCL:
   #_w1 := "E22" AND NOT "DB01_Osr".osr1;   // rising edge
   "DB01_Osr".osr1 := "E22";
   IF #_w1 THEN "DB03_Machine".dbw12 := "DB03_Machine".dbw12 - 1; END_IF;
END_REGION

REGION Network 29: Counter for revolution on running height
   RUNG wire#powerrail
      I_Contact( "M0.5" )
      { S7_GenerateENO := "TRUE" } Move(in := "DB03_Machine".dbw76, out1 => "DB03_Machine".dbw12)
   END_RUNG
   // the same network as SCL:
   IF NOT "M0.5" THEN "DB03_Machine".dbw12 := "DB03_Machine".dbw76; END_IF;
END_REGION

REGION Network 30: Machine in wrapping cycle
   RUNG wire#powerrail
      Contact( "M0.1" )
      I_Contact( "On" )
      wire#w1
      S_SR(operand := "DB03_Machine".dbx7_5, r1 := wire#w2)
   END_RUNG
   RUNG wire#powerrail
      Contact( "M0.2" )
   END_RUNG wire#w1
   RUNG wire#powerrail
      Contact( "M0.0" )
   END_RUNG wire#w2
   RUNG wire#powerrail
      N_Contact(operand := "M1.4", bit := "M1.4_N")
   END_RUNG wire#w2
   // the same network as SCL:
   #_w1 := NOT "M1.4" AND "M1.4_N";   // falling edge of "M1.4"
   "M1.4_N" := "M1.4";
   IF ("M0.1" AND NOT "On") OR "M0.2" THEN
       "DB03_Machine".dbx7_5 := TRUE;   // SR flip-flop
   END_IF;
   IF "M0.0" OR #_w1 THEN "DB03_Machine".dbx7_5 := FALSE; END_IF;
END_REGION

REGION Network 31: Support memory to refresh pallet per hour value
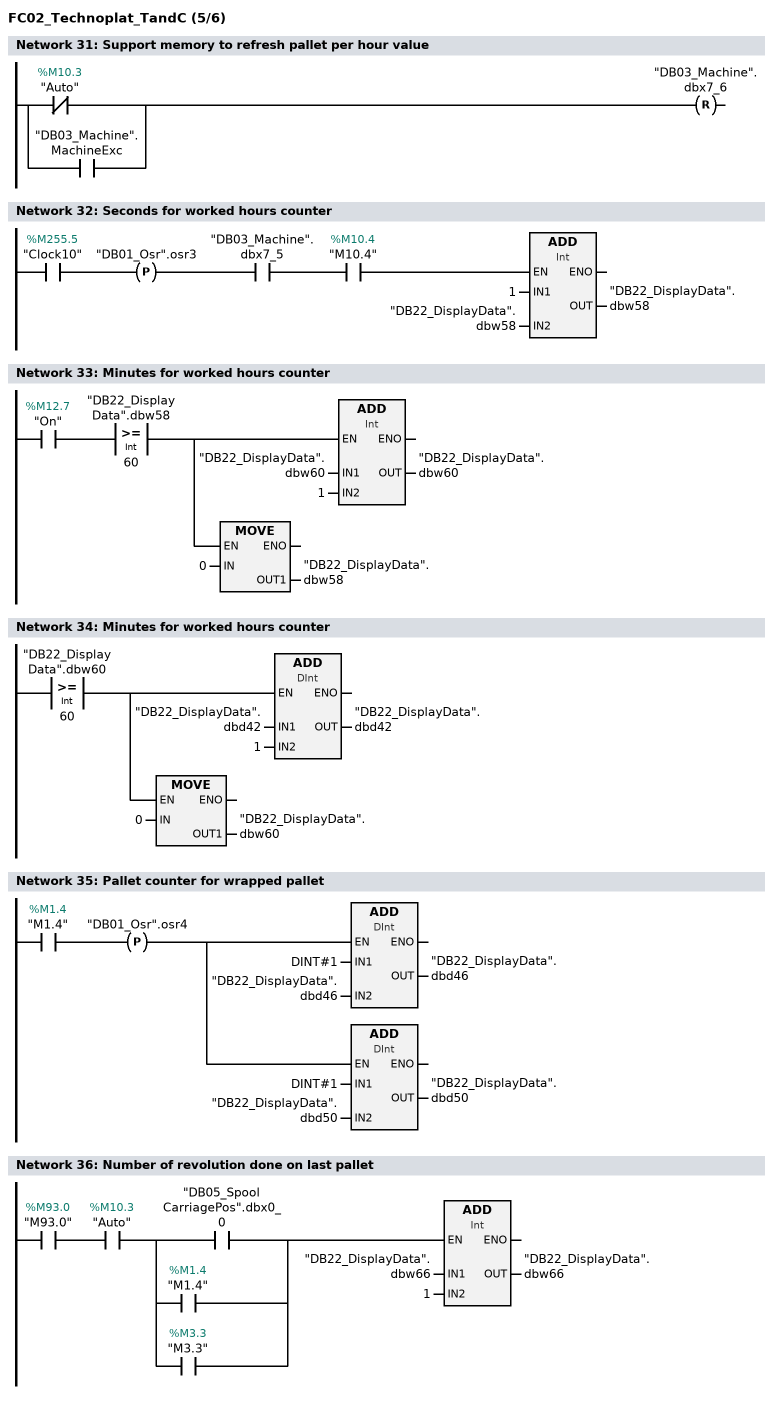
   RUNG wire#powerrail
      I_Contact( "Auto" )
      wire#w1
      R_Coil( "DB03_Machine".dbx7_6 )
   END_RUNG
   RUNG wire#powerrail
      Contact( "DB03_Machine".MachineExc )
   END_RUNG wire#w1
   // the same network as SCL:
   IF NOT "Auto" OR "DB03_Machine".MachineExc THEN "DB03_Machine".dbx7_6 := FALSE; END_IF;
END_REGION

REGION Network 32: Seconds for worked hours counter
   RUNG wire#powerrail
      Contact( "Clock10" )
      P_Trig( "DB01_Osr".osr3 )
      Contact( "DB03_Machine".dbx7_5 )
      Contact( "M10.4" )
      { S7_Templates := "SrcType := Int"; S7_GenerateENO := "TRUE" } Add(in1 := 1, in2 := "DB22_DisplayData".dbw58, out => "DB22_DisplayData".dbw58)
   END_RUNG
   // the same network as SCL:
   #_w1 := "Clock10" AND NOT "DB01_Osr".osr3;   // rising edge
   "DB01_Osr".osr3 := "Clock10";
   IF #_w1 AND "DB03_Machine".dbx7_5 AND "M10.4" THEN
       "DB22_DisplayData".dbw58 := 1 + "DB22_DisplayData".dbw58;
   END_IF;
END_REGION

REGION Network 33: Minutes for worked hours counter
   RUNG wire#powerrail
      Contact( "On" )
      { S7_Templates := "SrcType := Int" } GE_Contact(in1 := "DB22_DisplayData".dbw58, in2 := 60)
      wire#w1
      { S7_Templates := "SrcType := Int"; S7_GenerateENO := "TRUE" } Add(in1 := "DB22_DisplayData".dbw60, in2 := 1, out => "DB22_DisplayData".dbw60)
   END_RUNG
   RUNG wire#w1
      { S7_GenerateENO := "TRUE" } Move(in := 0, out1 => "DB22_DisplayData".dbw58)
   END_RUNG
   // the same network as SCL:
   IF "On" AND ("DB22_DisplayData".dbw58 >= 60) THEN
       "DB22_DisplayData".dbw60 := "DB22_DisplayData".dbw60 + 1;
       "DB22_DisplayData".dbw58 := 0;
   END_IF;
END_REGION

REGION Network 34: Minutes for worked hours counter
   RUNG wire#powerrail
      { S7_Templates := "SrcType := Int" } GE_Contact(in1 := "DB22_DisplayData".dbw60, in2 := 60)
      wire#w1
      { S7_Templates := "SrcType := DInt"; S7_GenerateENO := "TRUE" } Add(in1 := "DB22_DisplayData".dbd42, in2 := 1, out => "DB22_DisplayData".dbd42)
   END_RUNG
   RUNG wire#w1
      { S7_GenerateENO := "TRUE" } Move(in := 0, out1 => "DB22_DisplayData".dbw60)
   END_RUNG
   // the same network as SCL:
   IF "DB22_DisplayData".dbw60 >= 60 THEN
       "DB22_DisplayData".dbd42 := "DB22_DisplayData".dbd42 + 1;
       "DB22_DisplayData".dbw60 := 0;
   END_IF;
END_REGION

REGION Network 35: Pallet counter for wrapped pallet
   RUNG wire#powerrail
      Contact( "M1.4" )
      P_Trig( "DB01_Osr".osr4 )
      wire#w1
      { S7_Templates := "SrcType := DInt"; S7_GenerateENO := "TRUE" } Add(in1 := DINT#1, in2 := "DB22_DisplayData".dbd46, out => "DB22_DisplayData".dbd46)
   END_RUNG
   RUNG wire#w1
      { S7_Templates := "SrcType := DInt"; S7_GenerateENO := "TRUE" } Add(in1 := DINT#1, in2 := "DB22_DisplayData".dbd50, out => "DB22_DisplayData".dbd50)
   END_RUNG
   // the same network as SCL:
   #_w1 := "M1.4" AND NOT "DB01_Osr".osr4;   // rising edge
   "DB01_Osr".osr4 := "M1.4";
   IF #_w1 THEN
       "DB22_DisplayData".dbd46 := DINT#1 + "DB22_DisplayData".dbd46;
       "DB22_DisplayData".dbd50 := DINT#1 + "DB22_DisplayData".dbd50;
   END_IF;
END_REGION

REGION Network 36: Number of revolution done on last pallet
   RUNG wire#powerrail
      Contact( "M93.0" )
      Contact( "Auto" )
      wire#w1
      Contact( "DB05_SpoolCarriagePos".dbx0_0 )
      wire#w2
      { S7_Templates := "SrcType := Int"; S7_GenerateENO := "TRUE" } Add(in1 := "DB22_DisplayData".dbw66, in2 := 1, out => "DB22_DisplayData".dbw66)
   END_RUNG
   RUNG wire#w1
      Contact( "M1.4" )
   END_RUNG wire#w2
   RUNG wire#w1
      Contact( "M3.3" )
   END_RUNG wire#w2
   // the same network as SCL:
   IF "M93.0" AND "Auto" AND ("DB05_SpoolCarriagePos".dbx0_0 OR "M1.4" OR "M3.3") THEN
       "DB22_DisplayData".dbw66 := "DB22_DisplayData".dbw66 + 1;
   END_IF;
END_REGION

REGION Network 37: Number of revolution done on last pallet
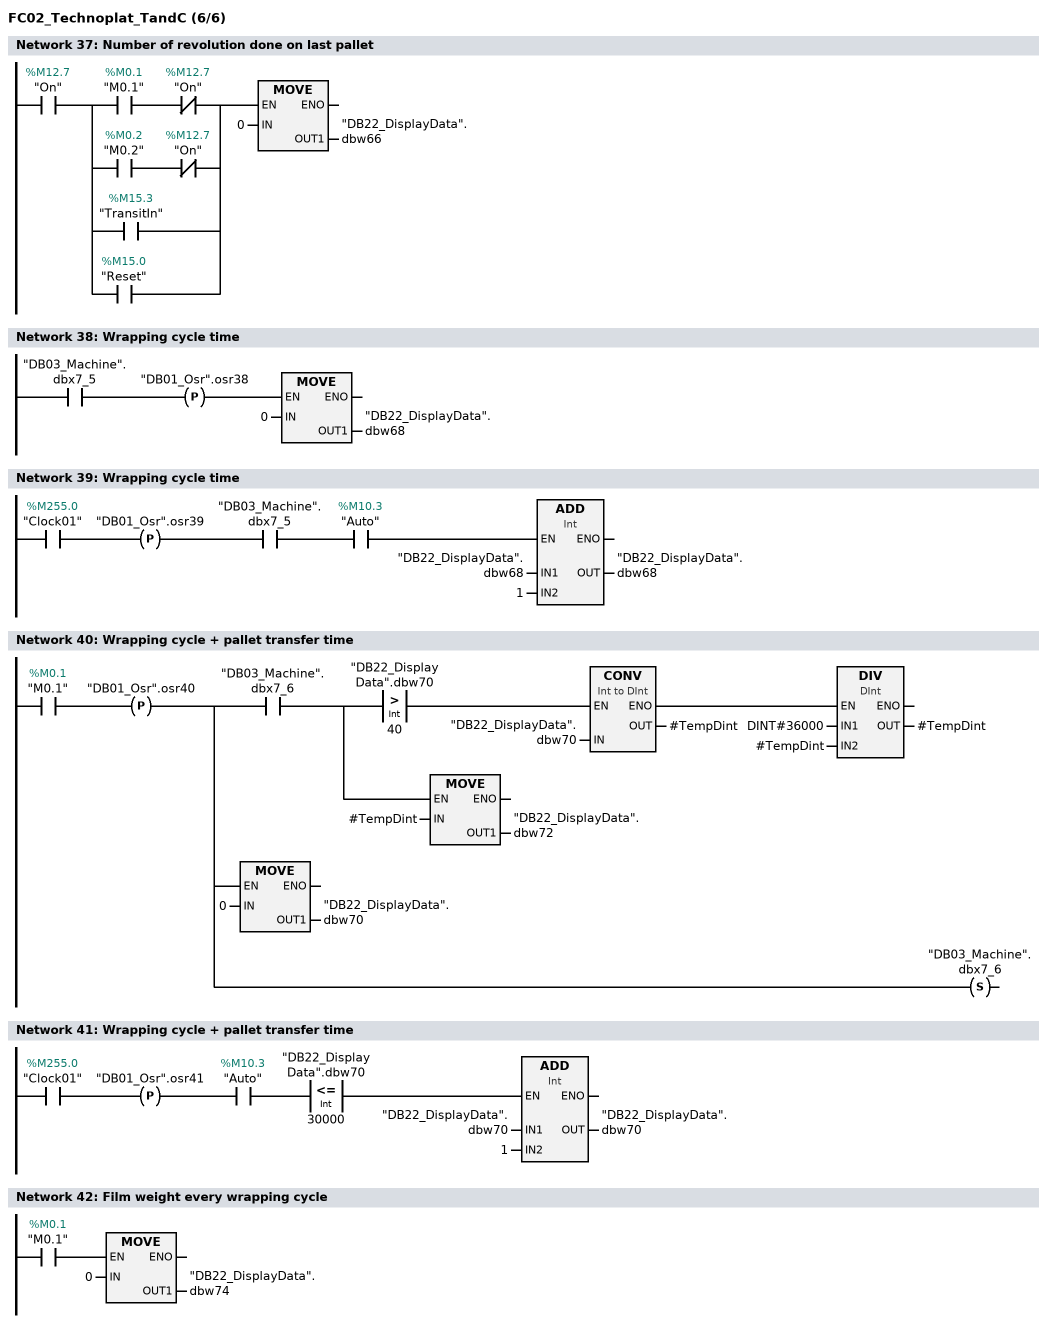
   RUNG wire#powerrail
      Contact( "On" )
      wire#w1
      Contact( "M0.1" )
      I_Contact( "On" )
      wire#w2
      { S7_GenerateENO := "TRUE" } Move(in := 0, out1 => "DB22_DisplayData".dbw66)
   END_RUNG
   RUNG wire#w1
      Contact( "M0.2" )
      I_Contact( "On" )
   END_RUNG wire#w2
   RUNG wire#w1
      Contact( "TransitIn" )
   END_RUNG wire#w2
   RUNG wire#w1
      Contact( "Reset" )
   END_RUNG wire#w2
   // the same network as SCL:
   IF "On" AND (("M0.1" AND NOT "On") OR ("M0.2" AND NOT "On") OR "TransitIn" OR "Reset") THEN
       "DB22_DisplayData".dbw66 := 0;
   END_IF;
END_REGION

REGION Network 38: Wrapping cycle time
   RUNG wire#powerrail
      Contact( "DB03_Machine".dbx7_5 )
      P_Trig( "DB01_Osr".osr38 )
      { S7_GenerateENO := "TRUE" } Move(in := 0, out1 => "DB22_DisplayData".dbw68)
   END_RUNG
   // the same network as SCL:
   #_w1 := "DB03_Machine".dbx7_5 AND NOT "DB01_Osr".osr38;   // rising edge
   "DB01_Osr".osr38 := "DB03_Machine".dbx7_5;
   IF #_w1 THEN "DB22_DisplayData".dbw68 := 0; END_IF;
END_REGION

REGION Network 39: Wrapping cycle time
   RUNG wire#powerrail
      Contact( "Clock01" )
      P_Trig( "DB01_Osr".osr39 )
      Contact( "DB03_Machine".dbx7_5 )
      Contact( "Auto" )
      { S7_Templates := "SrcType := Int"; S7_GenerateENO := "TRUE" } Add(in1 := "DB22_DisplayData".dbw68, in2 := 1, out => "DB22_DisplayData".dbw68)
   END_RUNG
   // the same network as SCL:
   #_w1 := "Clock01" AND NOT "DB01_Osr".osr39;   // rising edge
   "DB01_Osr".osr39 := "Clock01";
   IF #_w1 AND "DB03_Machine".dbx7_5 AND "Auto" THEN
       "DB22_DisplayData".dbw68 := "DB22_DisplayData".dbw68 + 1;
   END_IF;
END_REGION

REGION Network 40: Wrapping cycle + pallet transfer time
   RUNG wire#powerrail
      Contact( "M0.1" )
      P_Trig( "DB01_Osr".osr40 )
      wire#w1
      Contact( "DB03_Machine".dbx7_6 )
      wire#w2
      { S7_Templates := "SrcType := Int" } GT_Contact(in1 := "DB22_DisplayData".dbw70, in2 := 40)
      { S7_Templates := "[SrcType := Int, DestType := DInt]"; S7_GenerateENO := "TRUE" } Convert(in := "DB22_DisplayData".dbw70, out => #TempDint)
      { S7_Templates := "SrcType := DInt"; S7_GenerateENO := "TRUE" } Div(in1 := DINT#36000, in2 := #TempDint, out => #TempDint)
   END_RUNG
   RUNG wire#w2
      { S7_GenerateENO := "TRUE" } Move(in := #TempDint, out1 => "DB22_DisplayData".dbw72)
   END_RUNG
   RUNG wire#w1
      { S7_GenerateENO := "TRUE" } Move(in := 0, out1 => "DB22_DisplayData".dbw70)
   END_RUNG
   RUNG wire#w1
      S_Coil( "DB03_Machine".dbx7_6 )
   END_RUNG
   // the same network as SCL:
   // ENO of a box is taken as its EN; it also drops when the box reports an error
   #_w1 := "M0.1" AND NOT "DB01_Osr".osr40;   // rising edge
   "DB01_Osr".osr40 := "M0.1";
   #_w2 := #_w1 AND "DB03_Machine".dbx7_6;
   IF #_w2 AND ("DB22_DisplayData".dbw70 > 40) THEN
       #TempDint := INT_TO_DINT("DB22_DisplayData".dbw70);
       #TempDint := DINT#36000 / #TempDint;
   END_IF;
   IF #_w2 THEN "DB22_DisplayData".dbw72 := #TempDint; END_IF;
   IF #_w1 THEN
       "DB22_DisplayData".dbw70 := 0;
       "DB03_Machine".dbx7_6 := TRUE;
   END_IF;
END_REGION

REGION Network 41: Wrapping cycle + pallet transfer time
   RUNG wire#powerrail
      Contact( "Clock01" )
      P_Trig( "DB01_Osr".osr41 )
      Contact( "Auto" )
      { S7_Templates := "SrcType := Int" } LE_Contact(in1 := "DB22_DisplayData".dbw70, in2 := 30000)
      { S7_Templates := "SrcType := Int"; S7_GenerateENO := "TRUE" } Add(in1 := "DB22_DisplayData".dbw70, in2 := 1, out => "DB22_DisplayData".dbw70)
   END_RUNG
   // the same network as SCL:
   #_w1 := "Clock01" AND NOT "DB01_Osr".osr41;   // rising edge
   "DB01_Osr".osr41 := "Clock01";
   IF #_w1 AND "Auto" AND ("DB22_DisplayData".dbw70 <= 30000) THEN
       "DB22_DisplayData".dbw70 := "DB22_DisplayData".dbw70 + 1;
   END_IF;
END_REGION

REGION Network 42: Film weight every wrapping cycle
   RUNG wire#powerrail
      Contact( "M0.1" )
      { S7_GenerateENO := "TRUE" } Move(in := 0, out1 => "DB22_DisplayData".dbw74)
   END_RUNG
   // the same network as SCL:
   IF "M0.1" THEN "DB22_DisplayData".dbw74 := 0; END_IF;
END_REGION
END_FUNCTION

FUNCTION "FC03_TechnoplatAux" : Void   // FC3, LAD
TITLE = Auxiliary memory for the machine
{ S7_Optimized_Access := 'FALSE' }
AUTHOR : Robopac
VERSION : 0.0
// stored: AutoNumber false, IsIECCheckEnabled false, SetENOAutomatically false, UDAEnableTagReadback false
   VAR_INPUT
      PHASE : Bool;
   END_VAR
   VAR_TEMP
      Pulse_Reset : Bool;   // Pulse to reset encoders
      SuppSpeed : DWord;
      TempInt_min : Int;
      TempInt_max : Int;
      TempDint : DInt;
   END_VAR
   VAR_TEMP   // added for the SCL form of the ladder/FBD networks
      _w1 : Bool;
      _w2 : Bool;
      _w3 : Bool;
      _w4 : Bool;
   END_VAR
BEGIN

REGION Network 1: OSR and OSF for table phases sensor
